// TwinCAT 3 PLC project Tc_Devices
// Title: Tc_Devices
// Company: NewEngineer
// Author: https://github.com/phucpha
// ProjectVersion: 3.2.3.0
// Description: this library use for all Real devices without require special license.
// ProgramVersion: 3.1.4024.0
// libraries:
//   Tc2_Standard, * (Beckhoff Automation GmbH)
//   Tc2_System, * (Beckhoff Automation GmbH)
//   Tc3_Module, * (Beckhoff Automation GmbH)
//   Tc_Utilities, * (NewEngineer)
// project tree:
//   DUTs/ActivePower/ E_ActivePowerType.TcDUT
//   DUTs/Burner/ E_EcoFlamState.TcDUT, E_EcoFlamStateResetV3.TcDUT
//   DUTs/Contactor/ E_ContactorError.TcDUT, E_ContactorState.TcDUT, E_ContactorStateGo.TcDUT
//   DUTs/Cylinder/Universal Cylinder/ E_CylinderError.TcDUT, E_CylinderState.TcDUT, E_CylinderStateGo.TcDUT (not stored)
//   DUTs/Digital Devices/Digital Input/ E_DigitalInputExState.TcDUT (not stored)
//   DUTs/Digital Devices/Lamp Indicator/ E_LampState.TcDUT
//   DUTs/Tank/ E_TankState.TcDUT
//   DUTs/Visu/Burner/ E_VisuCtrlBurnerState.TcDUT, ST_VisuCtrlBurnerFrame.TcDUT
//   DUTs/Visu/Cylinder/ E_VisuCtrlCylinderImgType.TcDUT (not stored), E_VisuCtrlSingleCylinderState.TcDUT (not stored), ST_VisuCtrlCylinderFrame.TcDUT
//   DUTs/Visu/DIDO/ ST_VisuCtrlInputFrame.TcDUT, ST_VisuCtrlOutputFrame.TcDUT
//   / GlobalTextList.TcGTLO, PlcTask.TcTTO
//   POUs/ActivePower/ I_ActivePower.TcIO, I_ActivePowerNoFB.TcIO
//   POUs/AnalogIn/ FB_AnalogInputThermocouple.TcPOU
//   POUs/BurnerEcoflam/ FB_BurnerControlEcoFlam.TcPOU, FB_BurnerControlEcoFlamV2.TcPOU, FB_BurnerControlEcoFlamV3.TcPOU, I_BurnerControlEcoFlam.TcIO, I_BurnerControlEcoFlamV2.TcIO, I_BurnerControlEcoFlamV3.TcIO
//   POUs/ContactorTherRelay/ FB_Contactor1FB_ThermalRelay.TcPOU, FB_ContactorNonFB_Flex_ThermalRelay.TcPOU, FB_ContactorNonFB_ThermalRelay.TcPOU
//   POUs/Contactor/ FB_ContactorFBNO.TcPOU, FB_ContactorNonFB_Flex.TcPOU, FB_ContactorNonFB.TcPOU
//   POUs/Cylinder/Double Coil Cylinder/ FB_DoubleCoilCylinder.TcPOU (not stored)
//   POUs/Cylinder/Single Coil Cylinder/ FB_SingleCoilCylinder.TcPOU (not stored)
//   POUs/Cylinder/Universal Cylinder/ FB_UniversalCylinder.TcPOU, I_UniversalCylinder.TcIO (not stored)
//   POUs/Digital Devices/Digital Device/ FB_DigitalDevice.TcPOU, I_DigitalDevice.TcIO (not stored)
//   POUs/Digital Devices/Digital Input/ FB_DigitalInput.TcPOU, FB_DigitalInputExt.TcPOU, I_DigitalInput.TcIO (not stored)
//   POUs/Digital Devices/Digital Output/ FB_DigitalOutput.TcPOU, I_DigitalOutput.TcIO (not stored)
//   POUs/Digital Devices/Lamp Indicator/ FB_Lamp.TcPOU, I_Lamp.TcIO (not stored)
//   POUs/ POU.TcPOU
//   POUs/Tank0FB/ FB_SingleTankSV1Ext.TcPOU, FB_SingleTankSV1.TcPOU, FB_SingleTankS.TcPOU
//   POUs/TankFB/ FB_SingleTank.TcPOU (not stored), FB_SingleTankV0.TcPOU, FB_SingleTankV1.TcPOU, FB_TankFourCompartments.TcPOU
//   POUs/TankFB/Fill/ FB_TankFill_2Cylinder.TcPOU, I_TankFill.TcIO
//   POUs/TankMix/ FB_Mixer0.TcPOU
//   VISUs/Image Pools/ IPCylinder.TcIPO (not stored)
//   VISUs/Pages/ PageManualCylinders.TcVIS, PageManualInputs.TcVIS, PageManualOutputs.TcVIS, PageManualSafety.TcVIS
//   VISUs/Single/ SingleCylinder.TcVIS, SingleDigitalInput.TcVIS, SingleDigitalOutput.TcVIS, SingleSafeInput.TcVIS, SingleSafeOutput.TcVIS
//   VISUs/Text Lists/ TL_SingleCylinderState.TcTLO
// real-time tasks:
//   TASK PlcTask: cycle T#10ms, priority 20, ADS port 350

CONFIGURATION Tc_Devices
    RESOURCE PLC ON TwinCAT3
        TASK PlcTask(INTERVAL := T#10ms, PRIORITY := 20);
        PROGRAM POU WITH PlcTask : POU;
    END_RESOURCE
END_CONFIGURATION

// ---- DUTs/ActivePower/E_ActivePowerType.TcDUT
{attribute 'strict'}
TYPE E_ActivePowerType :
(
	ACTIVE_POWER_TYPE_NO_FEEDBACK,
	ACTIVE_POWER_TYPE_FEEDBACK
);
END_TYPE

// ---- DUTs/Burner/E_EcoFlamState.TcDUT
{attribute 'strict'}
{attribute 'to_string'}
TYPE E_EcoFlamState :
(
	ECOFLAM_ABORTING := -50,
	ECOFLAM_UNINITIALIZED := 0,
	ECOFLAM_INITIALIZING := 10,
	ECOFLAM_READY_INITIALIZED := 20,
	ECOFLAM_IGNITION := 30,
	ECOFLAM_IGNITION_DONE := 40,
	ECOFLAM_STOP := 50,
	ECOFLAM_STOP_DONE := 60,
	ECOFLAM_RESET := 70,
	ECOFLAM_RESET_DONE := 80
);
END_TYPE

// ---- DUTs/Burner/E_EcoFlamStateResetV3.TcDUT
{attribute 'strict'}
TYPE E_EcoFlamStateResetV3 :
(
	ECOFLAM_V3_RESET_TURN_OFF,
	ECOFLAM_V3_RESET_TURN_ON,
	ECOFLAM_V3_RESET_PORESET_ON
);
END_TYPE

// ---- DUTs/Contactor/E_ContactorError.TcDUT
{attribute 'strict'}
{Attribute 'to_string'}
TYPE E_ContactorError :
(
	CONTACTOR_ERROR_OK := 0,
	CONTACTOR_ERROR_POWER_ON_TIMED_OUT := 20
)UDINT := CONTACTOR_ERROR_OK;
END_TYPE

// ---- DUTs/Contactor/E_ContactorState.TcDUT
{attribute 'strict'}
{Attribute 'to_string'}
TYPE E_ContactorState :
(
	CONTACTOR_ABORTING 			:= -10,
	CONTACTOR_UNINITIALIZED		:= 0,	
	CONTACTOR_INITIALIZING		:= 10,	
	CONTACTOR_READY_INITIALIZED	:= 20,	
	CONTACTOR_IDLE				:= 30,	
	CONTACTOR_POWER_ON			:= 40,
	CONTACTOR_POWER_ON_DONE		:= 50,
	CONTACTOR_POWER_OFF			:= 60,
	CONTACTOR_POWER_OFF_DONE	:= 70,
	CONTACTOR_RESET				:= 100,
	CONTACTOR_RESET_DONE		:= 110

);
END_TYPE

// ---- DUTs/Contactor/E_ContactorStateGo.TcDUT
{Attribute 'to_string'}
{attribute 'strict'}
TYPE E_ContactorStateGo :
(
	CONTACTOR_MOVE_START_TRACKING	:= 0,
	CONTACTOR_MOVE_DELAY			:= 10,
	CONTACTOR_MOVE_DONE				:= 20
);
END_TYPE

// ---- DUTs/Cylinder/Universal Cylinder/E_CylinderError.TcDUT
{attribute 'strict'}
{attribute 'to_string'}
TYPE E_CylinderError :
(
	CYLINDER_ERROR_OK						:= 0,	(*  *)
	CYLINDER_ERROR_MOVE_HOME_TIMED_OUT 		:= 10,	(*  *)
	CYLINDER_ERROR_MOVE_ACTIVE_TIMED_OUT 	:= 20	(*  *)
);
END_TYPE

// ---- DUTs/Cylinder/Universal Cylinder/E_CylinderState.TcDUT
{attribute 'strict'}
{attribute 'to_string'}
TYPE E_CylinderState :
(
	CYLINDER_UNINITIALIZED		:= 0,	(* Cylinder is uninitialized *)
	CYLINDER_INITIALIZING		:= 10,	(* Initialization in progress *)
	CYLINDER_READY_INITIALIZED	:= 20,	(*  *)
	CYLINDER_IDLE				:= 30,	(* Cylinder ready to work *)
	CYLINDER_GO_ACTIVE			:= 40,	(* Cylinder is going to active position *)
	CYLINDER_GO_ACTIVE_DONE		:= 50,	(* Cylinder is in active position *)
	CYLINDER_GO_HOME			:= 60,	(* Cylinder is going to home position *)
	CYLINDER_GO_HOME_DONE		:= 70,	(* Cylinder is in home position *)
	CYLINDER_RELEASE			:= 80,	(* Cylinder is going to release all valves *)
	CYLINDER_RELEASE_DONE		:= 90,	(* Cylinder has been released *)
	CYLINDER_RESET				:= 100,	(* Reseting function block *)
	CYLINDER_RESET_DONE			:= 110,	(* Reset done *)
	CYLINDER_ABORTING 			:= -10	(* Aborting *)
);
END_TYPE

// ---- DUTs/Digital Devices/Lamp Indicator/E_LampState.TcDUT
{attribute 'strict'}
{Attribute 'to_string'}
TYPE E_LampState :
(
	LAMP_OFF 			:= 0,	(* Lamp is off *)
	LAMP_ON				:= 10,	(* Lamp is on *)
	LAMP_BLINKING_OFF	:= 20,	(* Lamp is blinking - current off *)
	LAMP_BLINKING_ON	:= 30	(* Lamp is bliniking - current on *)
);
END_TYPE

// ---- DUTs/Tank/E_TankState.TcDUT
TYPE E_TankState :
(	TANK_IDLE := 0,
	TANK_STOP := 5,
	TANK_WITHDRAWING := 10,
	TANK_WITHDRAWING_DONE := 15,
	TANK_FILLING:= 20
);
END_TYPE

// ---- DUTs/Visu/Burner/E_VisuCtrlBurnerState.TcDUT
{attribute 'strict'}
TYPE E_VisuCtrlBurnerState :
(
	VISU_CTRL_BURNER_WAIT_FOR_CMD 		:= 0,	(* *)
	VISU_CTRL_BURNER_INIT				:= 10,	(*  *)
	VISU_CTRL_BURNER_RESET				:= 20,	(*  *)
	VISU_CTRL_BURNER_IGNITION			:= 30,	(*  *)
	VISU_CTRL_BURNER_STOP				:= 40,	(*  *)
	VISU_CTRL_BURNER_APPEND_POWER_ON	:= 50,	(*  *)	
	VISU_CTRL_BURNER_ABORT				:= -10	(*  *)
);
END_TYPE

// ---- DUTs/Visu/Burner/ST_VisuCtrlBurnerFrame.TcDUT
TYPE ST_VisuCtrlBurnerFrame :
STRUCT
	btnInit				: BOOL;
	btnReset			: BOOL;
	btnAbort			: BOOL;
	btnAppendPowerOn	: BOOL;
	btnIgnition			: BOOL;
	btnStop				: BOOL;
	sName				: STRING;
	bError				: BOOL;
	bFault				: BOOL;
	bIgnitionSuccess	: BOOL;
	
	eState				: E_EcoFlamState;
	sState				: STRING;
END_STRUCT
END_TYPE

// ---- DUTs/Visu/Cylinder/ST_VisuCtrlCylinderFrame.TcDUT
TYPE ST_VisuCtrlCylinderFrame:
STRUCT
	sName			: STRING;
	btnInit				: BOOL;				(*  *)
	btnAbort			: BOOL;				(*  *)
	btnReset			: BOOL;				(*  *)
	btnGoHome 			: BOOL;				(*  *)
	btnGoActive 		: BOOL;				(*  *)
	btnRealase 			: BOOL;				(*  *)
	
	bSensorHome 		: BOOL;				(*  *)
	bSensorActive 		: BOOL;				(*  *)
	bPositionHold		: BOOL;				(*  *)
	bError				: BOOL;				(*  *)
	iErrorID			: UDINT;			(*  *)
	
	tActiveMovement 	: TIME;				(*  *)
	tHomeMovement 		: TIME;				(*  *)
	
	sActiveDescription 	: STRING;			(*  *)
	sHomeDescription 	: STRING;			(*  *)
	sStateDescription	: STRING;			(*  *)
	
	sCylinderImage		: STRING;			(*  *)
	eCylinderState		: E_CylinderState;	(*  *)
	sCylinderState		: STRING;
END_STRUCT
END_TYPE

// ---- DUTs/Visu/DIDO/ST_VisuCtrlInputFrame.TcDUT
TYPE ST_VisuCtrlInputFrame:
STRUCT
	sName			: STRING;
	bIn				: BOOL;								(*  *)
	bForceIn		: BOOL;								(*  *)
	bForceDisabled	: BOOL	:=TRUE ;					(*  *)
	sModuleType		: STRING;							(* Module type e.g. EL1xxx *)
	sPortID			: STRING;							(* Wire id connected to port *)
END_STRUCT
END_TYPE

// ---- DUTs/Visu/DIDO/ST_VisuCtrlOutputFrame.TcDUT
TYPE ST_VisuCtrlOutputFrame:
STRUCT
	sName			: STRING;
	btnOut 			: BOOL; 		(* This button allows to control ouptu manualy if it's set as controlable *)
	bOut 			: BOOL;			(* This bit indicates the status of output in manual mode *)
	bControlable	: BOOL;			(* This bit is used to lock control of output via manual mode - read access only *)
	sModuleType		: STRING;		(* Module type e.g. EL1xxx *)
	sPortID			: STRING;		(* Wire id connected to port *)
END_STRUCT
END_TYPE

// ---- POUs/ActivePower/I_ActivePower.TcIO
INTERFACE I_ActivePower	// don't not EXTENDS I_ActivePowerNoFB, it violates Liskov Substitution Principle (LSP)

PROPERTY Active : reference to bool
GET
END_GET
END_PROPERTY

PROPERTY Busy : REFERENCE TO bool
GET
END_GET
END_PROPERTY

PROPERTY Error : reference to bool
GET
END_GET
END_PROPERTY

METHOD MR_Abort : bool
VAR_INPUT
END_VAR
END_METHOD

METHOD MR_Init : bool
VAR_INPUT
END_VAR
END_METHOD

METHOD MR_PowerOFF : BOOL
VAR_INPUT
END_VAR
END_METHOD

METHOD MR_PowerON : BOOL
VAR_INPUT
END_VAR
END_METHOD

METHOD MR_Reset : bool
VAR_INPUT
END_VAR
END_METHOD

PROPERTY Name : STRING
GET
END_GET
SET
END_SET
END_PROPERTY

(*Powerer on success*)
PROPERTY Powered : REFERENCE TO BOOL
GET
END_GET
END_PROPERTY

PROPERTY PowerOffIsCalled : bool
GET
END_GET
END_PROPERTY

PROPERTY PowerOnIsCalled : bool
GET
END_GET
END_PROPERTY

(*return value depedning on Request*)
PROPERTY ReasonError : string
GET
END_GET
END_PROPERTY

END_INTERFACE

// ---- POUs/ActivePower/I_ActivePowerNoFB.TcIO
INTERFACE I_ActivePowerNoFB

METHOD MR_PowerOFF : BOOL
VAR_INPUT
END_VAR
END_METHOD

METHOD MR_PowerON : BOOL
VAR_INPUT
END_VAR
END_METHOD

PROPERTY Name : STRING
GET
END_GET
SET
END_SET
END_PROPERTY

PROPERTY PowerOffIsCalled : bool
GET
END_GET
END_PROPERTY

PROPERTY PowerOnIsCalled : bool
GET
END_GET
END_PROPERTY

END_INTERFACE

// ---- POUs/BurnerEcoflam/I_BurnerControlEcoFlam.TcIO
INTERFACE I_BurnerControlEcoFlam

PROPERTY Busy : reference to bool
GET
END_GET
END_PROPERTY

PROPERTY Error : REFERENCE to bool
GET
END_GET
END_PROPERTY

PROPERTY IgnitionSucess : bool
GET
END_GET
END_PROPERTY

PROPERTY Inited : bool
GET
END_GET
END_PROPERTY

PROPERTY IsStop : bool
GET
END_GET
END_PROPERTY

METHOD MR_Abort : BOOL
VAR_INPUT
END_VAR
END_METHOD

METHOD MR_AppendPowerOn : BOOL
VAR_INPUT
	iPowerON	: I_ActivePower;
END_VAR
END_METHOD

METHOD MR_Ignition : BOOL
VAR_INPUT
END_VAR
END_METHOD

METHOD  MR_Init : bool // just Acknowledge already append the I_activepower
VAR_INPUT
END_VAR
END_METHOD

METHOD MR_Reset : BOOL
VAR_INPUT
END_VAR
END_METHOD

METHOD MR_Stop : BOOL
VAR_INPUT
END_VAR
END_METHOD

PROPERTY Name : string
GET
END_GET
SET
END_SET
END_PROPERTY

PROPERTY Ref_IfActivePower : REFERENCE TO I_ActivePower
GET
END_GET
END_PROPERTY

PROPERTY Ref_piFault : reference to  FB_DigitalInput
GET
END_GET
END_PROPERTY

PROPERTY Ref_piIgnitionSucess : reference to  FB_DigitalInput
GET
END_GET
END_PROPERTY

PROPERTY State : E_EcoFlamState
GET
END_GET
END_PROPERTY

END_INTERFACE

// ---- POUs/BurnerEcoflam/I_BurnerControlEcoFlamV2.TcIO
INTERFACE I_BurnerControlEcoFlamV2 EXTENDS I_BurnerControlEcoFlam

PROPERTY Ref_poReset : REFERENCE TO fb_digitalOutput
GET
END_GET
END_PROPERTY

END_INTERFACE

// ---- POUs/BurnerEcoflam/I_BurnerControlEcoFlamV3.TcIO
INTERFACE I_BurnerControlEcoFlamV3 EXTENDS I_BurnerControlEcoFlamV2

PROPERTY Ref_poGasLv1 : REFERENCE TO FB_DigitalOutput
GET
END_GET
END_PROPERTY

PROPERTY Ref_poGasLv2 : REFERENCE TO FB_DigitalOutput
GET
END_GET
END_PROPERTY

PROPERTY Ref_poOnOff : REFERENCE TO FB_DigitalOutput
GET
END_GET
END_PROPERTY

END_INTERFACE

// ---- POUs/TankFB/Fill/I_TankFill.TcIO
INTERFACE I_TankFill

METHOD Close : BOOL
VAR_INPUT
END_VAR
END_METHOD

PROPERTY IsClose : bool
GET
END_GET
END_PROPERTY

PROPERTY IsOpen : bool
GET
END_GET
END_PROPERTY

METHOD Open : BOOL
VAR_INPUT
END_VAR
END_METHOD

END_INTERFACE

// ---- POUs/POU.TcPOU
PROGRAM POU
VAR
//	FB_BurnerControlEcoFlam : FB_BurnerControlEcoFlam;
//	FB_BurnerControlEcoFlamV2 : FB_BurnerControlEcoFlamV2;
//	FB_BurnerControlEcoFlamV3 : FB_BurnerControlEcoFlamV3;
//	FB_ContactorFBNO : FB_ContactorFBNO;
//	fb_contactorNonFB : FB_ContactorNonFB;
//	FB_Contactor1FB_ThermalRelay : FB_Contactor1FB_ThermalRelay;
//	FB_ContactorNonFB_ThermalRelay : FB_ContactorNonFB_ThermalRelay;
//	FB_ContactorNonFB_Flex_ThermalRelay : FB_ContactorNonFB_Flex_ThermalRelay;
//	FB_SingleCoilCylinder : FB_SingleCoilCylinder;
//	FB_DoubleCoilCylinder : FB_DoubleCoilCylinder;
//	fbsingletank : FB_SingleTank;
//	fbsingletankV0 : FB_SingleTankV0;
//	fbsingletankV1 : FB_SingleTankV1;
//	fbTankFourCompartments : FB_TankFourCompartments;
//	fbSingleTankV1 : FB_SingleTanksV1;
//	fbFillTank : FB_TankFill_2Cylinder;
//	fbMixer0 : FB_Mixer0;
 	//bIsClose : BOOL;
END_VAR

//fbSingleTankV1.AssignIfill(iFill := fbFillTank);
//bIsClose := fbsingletankV1.Ref_iFill.IsClose;

END_PROGRAM

// ---- POUs/AnalogIn/FB_AnalogInputThermocouple.TcPOU
FUNCTION_BLOCK FB_AnalogInputThermocouple EXTENDS FB_DigitalDevice// use for El 3314
VAR
	iRawValue	AT%I*: INT;
	lrSclale : LREAL := 0.1;
	lrValue	: LREAL;
	bError		AT%I* : BOOL;
	
END_VAR

lrValue := INT_TO_LREAL(iRawValue)*lrSclale;

PROPERTY Error :  bool
GET
Error := bError;
END_GET
END_PROPERTY

PROPERTY Scale : lreal // Value = rawValue form terminal * scale
GET
Scale := lrSclale;
END_GET
SET
lrSclale := Scale;
END_SET
END_PROPERTY

{attribute 'monitoring' := 'variable'}
PROPERTY Value : REFERENCE TO  lreal
GET
Value ref= lrValue;
END_GET
END_PROPERTY

END_FUNCTION_BLOCK

// ---- POUs/Digital Devices/Digital Device/FB_DigitalDevice.TcPOU
(* 
:Description: This function block is base for all other digital devices.
*)
FUNCTION_BLOCK ABSTRACT FB_DigitalDevice IMPLEMENTS I_DigitalDevice
VAR
	sName : STRING; (* Name of digital device instance *)
	sModuleType : STRING;
	sPortID		: STRING;
END_VAR

PROPERTY ModuleType : REFERENCE TO STRING
GET
ModuleType REF= sModuleType;
END_GET
END_PROPERTY

METHOD MR_FirstCycle : BOOL
VAR_INPUT
	sName : STRING;
	sModuleType : STRING;
	sPortID		: STRING;
END_VAR
THIS^.sName := sName;
THIS^.sModuleType := sModuleType;
THIS^.sPortID := sPortID;
END_METHOD

PROPERTY Name : REFERENCE TO STRING
GET
Name REF= sName;
END_GET
END_PROPERTY

PROPERTY PortID : REFERENCE TO STRING
GET
PortID REF= sPortID;
END_GET
END_PROPERTY

END_FUNCTION_BLOCK

// ---- POUs/BurnerEcoflam/FB_BurnerControlEcoFlam.TcPOU
(* This function use for BurnerControlEcoFlam
| this version dont have Reset components like Digital output, user have to reset manual at the BurnerControlEcoFlam device
*)
FUNCTION_BLOCK FB_BurnerControlEcoFlam IMPLEMENTS I_BurnerControlEcoFlam

VAR
	piFault	: FB_DigitalInput;
	piFireSussess : FB_DigitalInputExt;
	ifActivePower : I_ActivePower;					//have FB
	ifActivePowerNoFB : I_ActivePowerNoFB;
	eActivePowerType : E_ActivePowerType;
	eState	: E_EcoFlamState;
	bAbort: BOOL;
	bBusy: BOOL;
	bInit: BOOL;
	bReset: BOOL;
	bStop: BOOL;
	bError : BOOL;
	tMeasurement	: TIME := T#200S;
	bIgnition: BOOL;
	bIgnitioned: BOOL;
	tonMeasurementTimer: Ton;
	tBurnSuccess: TIME;
	sName : STRING;
END_VAR

bError := piFault.In; //OR piFireSussess.ErrorTimedout;
piFireSussess();
StateMachine();
tonMeasurementTimer(PT := tMeasurement);
IF piFireSussess.RisingTrigger AND eState = ECOFLAM_IGNITION THEN
	tBurnSuccess	:= 	tonMeasurementTimer.ET;				
END_IF

PROPERTY ActivePowerType : Reference to E_ActivePowerType
GET
ActivePowerType ref= eActivePowerType;
END_GET
END_PROPERTY

{attribute 'monitoring' := 'variable'}
PROPERTY Busy : reference to bool
GET
Busy ref= bBusy;
END_GET
END_PROPERTY

PROPERTY Error : REFERENCE to bool
GET
error REF= bError;
END_GET
END_PROPERTY

{attribute 'monitoring' := 'variable'}
PROPERTY IgnitionSucess : bool
GET
CASE eActivePowerType OF
	ACTIVE_POWER_TYPE_NO_FEEDBACK:
		IgnitionSucess := piFireSussess.In AND ifActivePowerNoFB.PowerOnIsCalled;
		
	ACTIVE_POWER_TYPE_FEEDBACK:
		IgnitionSucess := piFireSussess.In AND ifActivePower.PowerOnIsCalled;
END_CASE
END_GET
END_PROPERTY

PROPERTY Inited : bool
GET
Inited := eState=ECOFLAM_READY_INITIALIZED;
END_GET
END_PROPERTY

PROPERTY IsRefActivePower : bool
GET
IsRefActivePower := ifActivePower<>0 OR ifActivePowerNoFB<>0;
END_GET
END_PROPERTY

PROPERTY IsStop : bool
GET
CASE eActivePowerType OF
	ACTIVE_POWER_TYPE_NO_FEEDBACK:
		isStop := ifActivePowerNoFB.PowerOffIsCalled;
		
	ACTIVE_POWER_TYPE_FEEDBACK:
		isStop := NOT ifActivePower.Powered;
END_CASE
END_GET
END_PROPERTY

METHOD MR_Abort : BOOL
VAR_INPUT
END_VAR
IF eState >= ECOFLAM_INITIALIZING THEN
	bAbort := TRUE;
	bBusy := TRUE;
	MR_Abort := FALSE;
	eState := ECOFLAM_ABORTING;
ELSIF eState = ECOFLAM_UNINITIALIZED THEN
	bAbort := FALSE;
	bBusy := FALSE;
	MR_Abort := TRUE;
END_IF
END_METHOD

METHOD MR_AppendPowerOn : BOOL
VAR_INPUT
	iPowerON	: I_ActivePower;
END_VAR
IF THIS^.ifActivePower <> iPowerON THEN
	THIS^.ifActivePower := iPowerON;
	MR_AppendPowerOn := true;
END_IF
END_METHOD

METHOD MR_AppendPowerOnNoFB : BOOL
VAR_INPUT
	iPowerOnNoFB	: I_ActivePowerNoFB;
END_VAR
IF THIS^.ifActivePowerNoFB <> iPowerOnNoFB THEN
	THIS^.ifActivePowerNoFB := iPowerOnNoFB;
	MR_AppendPowerOnNoFB := true;
END_IF
END_METHOD

METHOD MR_ChooseIfActivePowerType : BOOL
VAR_INPUT
	eChoseActivePowerType : E_ActivePowerType;
END_VAR
eActivePowerType := eChoseActivePowerType;
END_METHOD

METHOD MR_FirstCycle : BOOL
VAR_INPUT
	sName 							: STRING;
	sPiFireSuccessModuleType		: STRING;
	sPiFirePortID					: STRING;
	sPiFaultModuleType				: STRING;
	sPiFaultPortID					: STRING;
	tONBurnerTimeOut				: TIME;
END_VAR
THIS^.sName := sName;
THIS^.piFireSussess.MR_FirstCycleEx(
 	sName			:= CONCAT(sName,':FireSuccess SS'),
	sModuleType 	:= sPiFireSuccessModuleType,
	sPortID			:= sPiFirePortID,
	bEnableTimeout	:= TRUE,
	tDefaultTimeout	:= tONBurnerTimeOut
);
										
THIS^.piFault.MR_FirstCycle(
	sName := CONCAT(sName,':Fault SS'),
	sModuleType := sPiFaultModuleType,
	sPortID := sPiFaultPortID
);
END_METHOD

METHOD MR_Ignition : BOOL
VAR_INPUT
END_VAR
CASE eActivePowerType OF
	ACTIVE_POWER_TYPE_NO_FEEDBACK:
		IF eState = ECOFLAM_READY_INITIALIZED AND NOT ifActivePowerNoFB.PowerOnIsCalled THEN
			bIgnition	:= TRUE;
			MR_Ignition := FALSE;
			bIgnitioned	:= FALSE;
			eState := ECOFLAM_IGNITION;
			bBusy := TRUE;
		ELSIF eState = ECOFLAM_IGNITION_DONE THEN
			bIgnition := FALSE;
			bIgnitioned	:= TRUE;
			MR_Ignition := TRUE;
			bBusy := false	;
		END_IF
		
	ACTIVE_POWER_TYPE_FEEDBACK:
		IF eState = ECOFLAM_READY_INITIALIZED AND NOT ifActivePower.PowerOnIsCalled THEN
			bIgnition	:= TRUE;
			MR_Ignition := FALSE;
			bIgnitioned	:= FALSE;
			eState := ECOFLAM_IGNITION;
			bBusy := TRUE;
		ELSIF eState = ECOFLAM_IGNITION_DONE THEN
			bIgnition := FALSE;
			bIgnitioned	:= TRUE;
			MR_Ignition := TRUE;
			bBusy := false	;
		END_IF
END_CASE
END_METHOD

METHOD  MR_Init : bool // just Acknowledge already append the I_activepower
VAR_INPUT
END_VAR
IF eState = ECOFLAM_UNINITIALIZED THEN
	bInit := TRUE;
	bBusy := TRUE;
	MR_Init := FALSE;
	eState := ECOFLAM_INITIALIZING;
ELSIF eState = ECOFLAM_READY_INITIALIZED THEN
	bInit := FALSE;
	MR_Init := TRUE;
	bBusy := false;
END_IF
END_METHOD

METHOD MR_Reset : BOOL
VAR_INPUT
END_VAR
IF eState >= ECOFLAM_READY_INITIALIZED AND bError THEN
	bBusy := TRUE;
	bReset := TRUE;
	MR_Reset := FALSE;
	eState := ECOFLAM_RESET;
ELSIF eState = ECOFLAM_RESET_DONE THEN
	bBusy := TRUE;
	bReset := FALSE;
	MR_Reset := TRUE;
END_IF
END_METHOD

METHOD MR_Stop : BOOL
VAR_INPUT
END_VAR
CASE eActivePowerType OF
	ACTIVE_POWER_TYPE_NO_FEEDBACK:
		IF eState >= ECOFLAM_INITIALIZING 
			AND eState < ECOFLAM_STOP_DONE 
			AND ifActivePowerNoFB.PowerOnIsCalled  
		THEN
			bStop := true;
			MR_Stop := FALSE;
			bBusy := TRUE;
			eState := ECOFLAM_STOP;
		ELSIF eState = ECOFLAM_STOP_DONE THEN
			bStop := FALSE;
			MR_Stop := TRUE;
			bBusy := false;
		END_IF 
		
	ACTIVE_POWER_TYPE_FEEDBACK:
		IF eState >= ECOFLAM_INITIALIZING 
			AND eState < ECOFLAM_STOP_DONE 
			AND ifActivePower.Powered  
		THEN
			bStop := true;
			MR_Stop := FALSE;
			bBusy := TRUE;
			eState := ECOFLAM_STOP;
		ELSIF eState = ECOFLAM_STOP_DONE THEN
			bStop := FALSE;
			MR_Stop := TRUE;
			bBusy := false;
		END_IF 
END_CASE
END_METHOD

METHOD PROTECTED  MS_Aborting
CASE eActivePowerType OF
	ACTIVE_POWER_TYPE_NO_FEEDBACK:
		ifActivePowerNoFB.MR_PowerOFF();
		piFireSussess.MR_Abort();
		IF NOT piFireSussess.Active THEN
			eState := ECOFLAM_UNINITIALIZED;
		END_IF
		
	ACTIVE_POWER_TYPE_FEEDBACK:
		ifActivePower.MR_PowerOFF();
		piFireSussess.MR_Abort();
		IF NOT ifActivePower.Powered 
			AND NOT ifActivePower.Busy 
			AND NOT piFireSussess.Active
		THEN
			eState := ECOFLAM_UNINITIALIZED;
		END_IF
END_CASE
END_METHOD

METHOD PROTECTED MS_Ignition
VAR_INPUT
END_VAR
CASE eActivePowerType OF
	ACTIVE_POWER_TYPE_NO_FEEDBACK:
		ifActivePowerNoFB.MR_PowerON();
		piFireSussess.MR_StartTracking();
		tonMeasurementTimer.IN := TRUE;
		IF piFireSussess.In  THEN
			eState := ECOFLAM_IGNITION_DONE;
		END_IF
		
	ACTIVE_POWER_TYPE_FEEDBACK:
		ifActivePower.MR_PowerON();
		piFireSussess.MR_StartTracking();
		tonMeasurementTimer.IN := TRUE;
		IF ifActivePower.Powered AND NOT ifActivePower.Busy 
		AND  piFireSussess.In  THEN
			eState := ECOFLAM_IGNITION_DONE;
		END_IF
END_CASE
END_METHOD

METHOD PROTECTED MS_IgnitionDone : BOOL
VAR_INPUT
END_VAR
tonMeasurementTimer.IN := false;
IF NOT bIgnition THEN
	eState :=  ECOFLAM_READY_INITIALIZED;
END_IF
END_METHOD

METHOD PROTECTED MS_Initializing
piFireSussess.MR_Init();
piFireSussess.EnableTimeout := TRUE;

CASE eActivePowerType OF
	ACTIVE_POWER_TYPE_NO_FEEDBACK:
		IF ifActivePowerNoFB <> 0
			AND piFireSussess.Active
		THEN
			eState := ECOFLAM_READY_INITIALIZED;
		END_IF
		
	ACTIVE_POWER_TYPE_FEEDBACK:
		IF ifActivePower <> 0
			AND piFireSussess.Active
		THEN
			eState := ECOFLAM_READY_INITIALIZED;
		END_IF
END_CASE
END_METHOD

METHOD PROTECTED MS_ReadyInitialized
VAR_INPUT
END_VAR
bBusy := false;
END_METHOD

(*
this version just reset piFireSussess, User have to reset manually at the device
*)
METHOD PROTECTED MS_Reset : BOOL
piFireSussess.MR_Reset();
bInit 		:= FALSE;
bAbort		:= FALSE;
bIgnition 	:= FALSE;
bStop 		:= FALSE;
IF NOT piFireSussess.ErrorTimedout THEN
	eState := ECOFLAM_RESET_DONE;
END_IF
END_METHOD

(* don't not edit*)
METHOD PROTECTED MS_ResetDone
VAR_INPUT
END_VAR
eState := ECOFLAM_READY_INITIALIZED;
END_METHOD

METHOD protected MS_Stop 
VAR_INPUT
END_VAR
CASE eActivePowerType OF
	ACTIVE_POWER_TYPE_NO_FEEDBACK:
		ifActivePowerNoFB.MR_PowerOFF();
		eState := ECOFLAM_STOP_DONE;
		
	ACTIVE_POWER_TYPE_FEEDBACK:
		ifActivePower.MR_PowerOFF();
		IF NOT ifActivePower.Powered AND not ifActivePower.Busy THEN
			eState := ECOFLAM_STOP_DONE;
		END_IF
END_CASE
END_METHOD

METHOD protected Ms_StopDone
VAR_INPUT
END_VAR
IF NOT bStop THEN
	eState := ECOFLAM_READY_INITIALIZED;
END_IF
END_METHOD

METHOD PROTECTED MS_Uninitialized
bBusy := FALSE;

piFireSussess.EnableForce := FALSE;
piFireSussess.EnableTimeout := FALSE;

bInit 		:= FALSE;
bReset		:= FALSE;
bAbort		:= FALSE;
END_METHOD

PROPERTY Name : string
GET
Name := sName;
END_GET
SET
sName := Name;
END_SET
END_PROPERTY

PROPERTY Ref_IfActivePower : REFERENCE TO I_ActivePower
GET
Ref_IfActivePower ref= ifActivePower;
END_GET
END_PROPERTY

PROPERTY Ref_IfActivePowerNoFB : REFERENCE TO I_ActivePowerNoFB
GET
Ref_IfActivePowerNoFB ref= ifActivePowerNoFB;
END_GET
END_PROPERTY

PROPERTY Ref_piFault : reference to  FB_DigitalInput
GET
ref_piFault ref= piFault;
END_GET
END_PROPERTY

PROPERTY Ref_piIgnitionSucess : reference to  FB_DigitalInput
GET
ref_piIgnitionSucess ref= piFireSussess;
END_GET
END_PROPERTY

PROPERTY State : E_EcoFlamState
GET
State := eState;
END_GET
END_PROPERTY

METHOD PROTECTED StateMachine
CASE eState OF
	ECOFLAM_UNINITIALIZED :
		MS_Uninitialized();
		
	ECOFLAM_INITIALIZING	:
		MS_Initializing();
		
	ECOFLAM_READY_INITIALIZED :
		MS_ReadyInitialized();
		
	ECOFLAM_IGNITION	:
		MS_Ignition();
		
	ECOFLAM_IGNITION_DONE	:
		MS_IgnitionDone();
		
	ECOFLAM_STOP		:
		MS_Stop();
		
	ECOFLAM_STOP_DONE	:
		Ms_StopDone();
		
	ECOFLAM_RESET:
		MS_Reset();
		
	ECOFLAM_RESET_DONE:
		MS_ResetDone();
		
	ECOFLAM_ABORTING :
		MS_Aborting();
	
END_CASE
END_METHOD

END_FUNCTION_BLOCK

// ---- POUs/Digital Devices/Digital Input/FB_DigitalInput.TcPOU
(* 
| :Description: This function block represents basic digital input and can be used for creating an instance of signle digital input device like buttons, switches, sensors.
| To get the current status of digital input use "Value" property. To simulate state of the input by software set "Enable Force" parameter and change value via "MR_ResetForceValue" and "MR_SetForceValue" methods.
*)
FUNCTION_BLOCK FB_DigitalInput EXTENDS FB_DigitalDevice IMPLEMENTS I_DigitalInput
VAR
	(* Internal status *)
	bIn				AT %I*	: BOOL;		(* Current value of input *)
	bInForced				: BOOL;		(* Forced value from software *)
	bEnableForce			: BOOL;		(* Enable forcing of the input from software *)
	bRisingTrigger 			: BOOL;		(* Rising trigger of input detected*)
	bFallingTrigger 		: BOOL;		(* Falling trigger of input detected*)
	
	(* Function blocks *)
	rtRisingTrigger 		: R_TRIG;	(* Rising trigger detecting FB*)
	ftFallingTrigger		: F_TRIG;	(* Falling trigger detecting FB*)
END_VAR

PROPERTY EnableForce : BOOL
GET
EnableForce := bEnableForce;
END_GET
SET
bEnableForce := EnableForce;
END_SET
END_PROPERTY

PROPERTY FallingTrigger : BOOL
GET
ftFallingTrigger(CLK := In, Q => bFallingTrigger);
FallingTrigger := bFallingTrigger;
END_GET
END_PROPERTY

PROPERTY In : BOOL
GET
IF NOT bEnableForce THEN
	In := bIn;
ELSE
	In := bInForced;
END_IF
END_GET
END_PROPERTY

METHOD MR_ResetForceValue
IF bEnableForce THEN
	bInForced := FALSE;
	
END_IF
END_METHOD

METHOD MR_SetForceValue
IF bEnableForce THEN
	bInForced := TRUE;
	
END_IF
END_METHOD

PROPERTY RisingTrigger : BOOL
GET
rtRisingTrigger(CLK := In, Q => bRisingTrigger);
RisingTrigger := bRisingTrigger;
END_GET
END_PROPERTY

END_FUNCTION_BLOCK

// ---- POUs/Digital Devices/Digital Input/FB_DigitalInputExt.TcPOU
(* 
| :Description: This function block represents basic digital input and can be used for creating an instance of signle digital input device like buttons, switches, sensors.
| To get the current status of digital input use "Value" property. To simulate state of the input by software set "Enable Force" parameter and change value via "MR_ResetForceValue" and "MR_SetForceValue" methods.
*)
FUNCTION_BLOCK FB_DigitalInputExt EXTENDS FB_DigitalInput
VAR
	(* Internal commands *)
	bInit 				: BOOL;		(*  *)
	bAbort				: BOOL;		(*  *)
	bReset				: BOOL;		(*  *)
	bTimeoutTracking	: BOOL;		(* Watchdog timer control bit *)
	
	(* Internal status *)
	bActive				: BOOL;		(*  *)
	bErrorTimedout		: BOOL;		(* Timeout coccured while waiting for signal *)
	eDigitalInputState	: E_DigitalInputExState;
	
	(*Internal parameters*)
	tTimeout			: TIME;		(* Input timeout *)
	bEnableTimeout		: BOOL;		(* Enable using timeout *)
	
	(* Function blocks *)
	bStartWatchdog		: BOOL;
	tonWatchdog			: TON;		(* Input timeout watchdog *)
	
END_VAR

bActive := eDigitalInputState >= DIGITAL_INPUT_EX_IDLE; //OR eDigitalInputState = DIGITAL_INPUT_EX_ABORTING;

StateMachine();

tonWatchdog( IN := bStartWatchdog, PT := tTimeout);

PROPERTY Active : REFERENCE TO BOOL
GET
Active REF= bActive;
END_GET
END_PROPERTY

PROPERTY CurrentTimeout : REFERENCE TO TIME
GET
CurrentTimeout REF= tonWatchdog.ET;
END_GET
END_PROPERTY

PROPERTY EnableTimeout : BOOL
GET
EnableTimeout := bEnableTimeout;
END_GET
SET
bEnableTimeout := EnableTimeout;
END_SET
END_PROPERTY

PROPERTY ErrorTimedout : REFERENCE TO BOOL
GET
ErrorTimedout REF= bErrorTimedout;
END_GET
END_PROPERTY

METHOD MR_Abort : BOOL
VAR_INPUT
END_VAR
IF eDigitalInputState > DIGITAL_INPUT_EX_UNINITIALIZED THEN
	bAbort := TRUE;
	MR_Abort := FALSE;
	eDigitalInputState := DIGITAL_INPUT_EX_ABORTING;
	fbMachineLogger.MR_AddLogs(CONCAT(sName,' : abort requested'));	
	
ELSIF eDigitalInputState = DIGITAL_INPUT_EX_UNINITIALIZED THEN
	bAbort := FALSE;
	MR_Abort := TRUE;
	fbMachineLogger.MR_AddLogs(CONCAT(sName,' : abort done'));	
	
END_IF
END_METHOD

METHOD MR_FirstCycleEx : BOOL
VAR_INPUT
	sName			: STRING;
	sModuleType		: STRING;
	sPortID			: STRING;
	bEnableTimeout	: BOOL;
	tDefaultTimeout : TIME;
END_VAR
THIS^.sName := sName;
THIS^.ModuleType := sModuleType;
THIS^.PortID := sPortID;
THIS^.bEnableTimeout := bEnableTimeout;
THIS^.tTimeout := tDefaultTimeout;
END_METHOD

METHOD MR_Init : BOOL
VAR_INPUT
END_VAR
IF eDigitalInputState = DIGITAL_INPUT_EX_UNINITIALIZED THEN
	bInit := TRUE;
	MR_Init := FALSE;
	eDigitalInputState := DIGITAL_INPUT_EX_INITIALIZING;
	fbMachineLogger.MR_AddLogs(CONCAT(sName,' : initialization requested'));		
	
ELSIF eDigitalInputState = DIGITAL_INPUT_EX_IDLE AND bInit THEN
	bInit := FALSE;
	MR_Init := TRUE;
	fbMachineLogger.MR_AddLogs(CONCAT(sName,' : initialization done'));	

END_IF
END_METHOD

METHOD MR_Reset : BOOL
VAR_INPUT
END_VAR
IF eDigitalInputState = DIGITAL_INPUT_EX_IDLE THEN
	bReset := TRUE;
	MR_Reset := FALSE;
	eDigitalInputState := DIGITAL_INPUT_EX_RESET;
	fbMachineLogger.MR_AddLogs(CONCAT(sName,' : reset requested'));	
	
ELSIF eDigitalInputState = DIGITAL_INPUT_EX_RESET_DONE THEN
	bReset := FALSE;
	MR_Reset := TRUE;
	fbMachineLogger.MR_AddLogs(CONCAT(sName,' : reset done'));	
	
END_IF
END_METHOD

METHOD MR_StartTracking
VAR_INPUT
END_VAR
IF eDigitalInputState = DIGITAL_INPUT_EX_IDLE AND bEnableTimeout AND NOT bErrorTimedout THEN
	bTimeoutTracking := TRUE;
	eDigitalInputState := DIGITAL_INPUT_EX_TIMEOUT_TRACKING;
	fbMachineLogger.MR_AddLogs(CONCAT(sName,' : start tracking requested'));	
	
END_IF
END_METHOD

METHOD PROTECTED MS_Abort
VAR_INPUT
END_VAR
eDigitalInputState := DIGITAL_INPUT_EX_UNINITIALIZED;
END_METHOD

METHOD PROTECTED MS_Idle
VAR_INPUT
END_VAR
;
END_METHOD

METHOD PROTECTED MS_Initializing
VAR_INPUT
END_VAR
(* To-Do add alarm declaration *)

eDigitalInputState := DIGITAL_INPUT_EX_READY_INITIALIZED;
END_METHOD

METHOD PROTECTED MS_ReadyInitialized
VAR_INPUT
END_VAR
eDigitalInputState := DIGITAL_INPUT_EX_IDLE;
END_METHOD

METHOD PROTECTED MS_Reset
VAR_INPUT
END_VAR
bErrorTimedout := FALSE;
eDigitalInputState := DIGITAL_INPUT_EX_RESET_DONE;
END_METHOD

METHOD PROTECTED MS_ResetDone
VAR_INPUT
END_VAR
IF NOT bReset THEN
	eDigitalInputState := DIGITAL_INPUT_EX_IDLE;
END_IF
END_METHOD

METHOD PROTECTED MS_TimeoutTracking
VAR_INPUT
END_VAR
IF tonWatchdog.Q THEN
	(* To-Do raise alarm *)
	bErrorTimedout := TRUE;
	bStartWatchdog := FALSE;
	eDigitalInputState := DIGITAL_INPUT_EX_TIMEOUT_TRACKING_DONE;
	
ELSE
	bStartWatchdog := TRUE;
	
	IF bRisingTrigger OR bFallingTrigger THEN
		bStartWatchdog := FALSE;
		eDigitalInputState := DIGITAL_INPUT_EX_TIMEOUT_TRACKING_DONE;
	
	END_IF
END_IF
END_METHOD

METHOD PROTECTED MS_TimeoutTrackingDone
VAR_INPUT
END_VAR
bTimeoutTracking := FALSE;
eDigitalInputState := DIGITAL_INPUT_EX_IDLE;
END_METHOD

METHOD PROTECTED MS_Uninitialized
VAR_INPUT
END_VAR
bInit := FALSE;
bAbort := FALSE;
bReset := FALSE;
bTimeoutTracking := FALSE;

bRisingTrigger := FALSE;
bFallingTrigger := FALSE;
bErrorTimedout := FALSE;

tonWatchdog( IN := FALSE, PT := tTimeout);
END_METHOD

PROPERTY State : REFERENCE TO E_DigitalInputExState
GET
State REF= eDigitalInputState;
END_GET
END_PROPERTY

METHOD PROTECTED StateMachine
VAR_INPUT
END_VAR
CASE eDigitalInputState OF
	DIGITAL_INPUT_EX_UNINITIALIZED:
		MS_Uninitialized();
		
	DIGITAL_INPUT_EX_INITIALIZING:
		MS_Initializing();
		
	DIGITAL_INPUT_EX_READY_INITIALIZED:
		MS_ReadyInitialized();
		
	DIGITAL_INPUT_EX_IDLE:
		MS_Idle();
		
	DIGITAL_INPUT_EX_TIMEOUT_TRACKING:
		MS_TimeoutTracking();	
	
	DIGITAL_INPUT_EX_TIMEOUT_TRACKING_DONE:
		MS_TimeoutTrackingDone();	
	
	DIGITAL_INPUT_EX_RESET:
		MS_Reset();

	DIGITAL_INPUT_EX_RESET_DONE:
		MS_ResetDone();
	
	DIGITAL_INPUT_EX_ABORTING:
		MS_Abort();
	
END_CASE
END_METHOD

PROPERTY Timeout : TIME
GET
Timeout := tTimeout;
END_GET
SET
tTimeout := Timeout;
END_SET
END_PROPERTY

END_FUNCTION_BLOCK

// ---- POUs/BurnerEcoflam/FB_BurnerControlEcoFlamV2.TcPOU
(* This function use for BurnerControlEcoFlam have Reset by Digital output.
*)
FUNCTION_BLOCK FB_BurnerControlEcoFlamV2 EXTENDS FB_BurnerControlEcoFlam IMPLEMENTS I_BurnerControlEcoFlamV2
VAR
	poReset : FB_DigitalOutput;
	tonReset : TON;
	timeReset : TIME := T#1.5s;
END_VAR

tonReset(
	in := eState=ECOFLAM_RESET,
	PT := timeReset
);
poReset();
poReset.Out := tonReset.IN;
SUPER^();

METHOD PROTECTED MS_Reset : BOOL
piFireSussess.MR_Reset();
bInit 		:= FALSE;
bAbort		:= FALSE;
bIgnition 	:= FALSE;
bStop 		:= FALSE;
IF NOT piFireSussess.ErrorTimedout// for sure least than TimeReset.
	AND tonReset.Q
THEN
	eState := ECOFLAM_RESET_DONE;
END_IF
END_METHOD

PROPERTY Ref_poReset : Reference to FB_DigitalOutput
GET
Ref_poReset ref= poReset;
END_GET
END_PROPERTY

END_FUNCTION_BLOCK

// ---- POUs/Digital Devices/Digital Output/FB_DigitalOutput.TcPOU
(* 
| :Description: This function block represents basic digital output and can be used for creating an instance of signle digital output device. 
| To control the output state use property "Out" 
*)
FUNCTION_BLOCK FB_DigitalOutput EXTENDS FB_DigitalDevice IMPLEMENTS  I_DigitalOutput
VAR
	bOut AT %Q*: BOOL; (* Current value of output*)
END_VAR

PROPERTY Out : BOOL
GET
Out := bOut;
END_GET
SET
bOut := Out;
END_SET
END_PROPERTY

END_FUNCTION_BLOCK

// ---- POUs/BurnerEcoflam/FB_BurnerControlEcoFlamV3.TcPOU
(* this fb for burner type that request off power and turn on again to reset it*)
FUNCTION_BLOCK FB_BurnerControlEcoFlamV3 EXTENDS FB_BurnerControlEcoFlamV2 IMPLEMENTS I_BurnerControlEcoFlamV3
VAR
	poOnOff : FB_DigitalOutput;
	poGasLv1 : FB_DigitalOutput;
	poGasLv2 : FB_DigitalOutput;
	eResetState : E_EcoFlamStateResetV3;
	tonDelayOffPower : TON;
	tonDelayOnPower : TON;
	timeDelayOnOffPower : TIME := T#2S;
END_VAR

IF IsRefActivePower THEN
	CASE ActivePowerType OF
		ACTIVE_POWER_TYPE_FEEDBACK:
			poOnOff.Out := ifActivePower.PowerOnIsCalled;
			poGasLv1.Out := ifActivePower.PowerOnIsCalled;
		ACTIVE_POWER_TYPE_NO_FEEDBACK:
			poOnOff.Out := ifActivePowerNoFB.PowerOnIsCalled;
			poGasLv1.Out := ifActivePowerNoFB.PowerOnIsCalled;
	END_CASE
END_IF
bError := piFault.In;
piFireSussess();
StateMachine();
tonMeasurementTimer(PT := tMeasurement);
IF piFireSussess.RisingTrigger AND eState=ECOFLAM_IGNITION THEN
	tBurnSuccess	:= 	tonMeasurementTimer.ET;				
END_IF

tonReset(
	in := (eState=ECOFLAM_RESET AND eResetState=ECOFLAM_V3_RESET_PORESET_ON),
	PT := timeReset
);
poReset();
poReset.Out := tonReset.IN;
tonDelayOffPower(
	IN := eState=ECOFLAM_RESET AND eresetstate=ECOFLAM_V3_RESET_TURN_OFF,
	PT := timeDelayOnOffPower
);
tonDelayOnPower(
	IN := eState=ECOFLAM_RESET AND eresetstate=ECOFLAM_V3_RESET_TURN_ON,
	PT := timeDelayOnOffPower
);

METHOD PROTECTED MS_Aborting
VAR_INPUT
END_VAR
SUPER^.MS_Aborting();
eResetState := ECOFLAM_V3_RESET_TURN_OFF;
END_METHOD

METHOD PROTECTED MS_Reset : BOOL
piFireSussess.MR_Reset();
bInit 		:= FALSE;
bAbort		:= FALSE;
bIgnition 	:= FALSE;
bStop 		:= FALSE;

CASE eResetState OF
	ECOFLAM_V3_RESET_TURN_OFF:
		CASE THIS^.eActivePowerType OF
			ACTIVE_POWER_TYPE_NO_FEEDBACK:
				ifActivePowerNoFB.MR_PowerOFF();
				IF tonDelayOffPower.Q THEN
					eResetState := ECOFLAM_V3_RESET_TURN_ON;
				END_IF
			ACTIVE_POWER_TYPE_FEEDBACK:
				ifActivePower.MR_PowerOFF();
				IF tonDelayOffPower.Q
					AND NOT ifActivePower.Powered AND NOT ifActivePower.Busy
				THEN
					eResetState := ECOFLAM_V3_RESET_TURN_ON;
				END_IF
		END_CASE
		
	ECOFLAM_V3_RESET_TURN_ON:
		CASE THIS^.eActivePowerType OF
			ACTIVE_POWER_TYPE_NO_FEEDBACK:
				ifActivePowerNoFB.MR_PowerON();
				IF tonDelayOnPower.Q THEN
					eResetState := ECOFLAM_V3_RESET_PORESET_ON;
				END_IF
			ACTIVE_POWER_TYPE_FEEDBACK:
				ifActivePower.MR_PowerON();
				IF (ifActivePower.Powered AND NOT ifActivePower.Busy)
					AND tonDelayOnPower.Q
				THEN
					eResetState := ECOFLAM_V3_RESET_PORESET_ON;
				END_IF
		END_CASE
		
	ECOFLAM_V3_RESET_PORESET_ON:
		IF tonReset.Q THEN
			eState := ECOFLAM_RESET_DONE;
		END_IF
END_CASE
END_METHOD

METHOD PROTECTED MS_ResetDone
VAR_INPUT
END_VAR
SUPER^.MS_ResetDone();
eResetState := ECOFLAM_V3_RESET_TURN_OFF;
END_METHOD

PROPERTY Ref_poGasLv1 : REFERENCE TO FB_DigitalOutput
GET
Ref_poGasLv1 ref= poGasLv1;
END_GET
END_PROPERTY

PROPERTY Ref_poGasLv2 : REFERENCE TO FB_DigitalOutput
GET
Ref_poGasLv2 ref= poGasLv2;
END_GET
END_PROPERTY

PROPERTY Ref_poOnOff : REFERENCE TO FB_DigitalOutput
GET
Ref_poOnOff ref= poOnOff;
END_GET
END_PROPERTY

END_FUNCTION_BLOCK

// ---- POUs/ContactorTherRelay/FB_Contactor1FB_ThermalRelay.TcPOU
(* 
| :Description: this function block is the Contactor FeedbackNO + thermal relay connect toghther.
| Then wiring have to series by Digital output to NC thermal relay to Coil
*)
FUNCTION_BLOCK FB_Contactor1FB_ThermalRelay EXTENDS FB_ContactorFBNO IMPLEMENTS I_ActivePower

VAR
	piFR		: FB_DigitalInput;// thermal relay NO
	bOverload	: BOOL;
END_VAR

bOverload :=  piFR.In;
SUPER^();

PROPERTY IsOverload : REFERENCE to bool
GET
isOverload ref= bOverload;
END_GET
END_PROPERTY

PROPERTY ReasonError : string
GET
IF isOverload THEN 
	ReasonError := 'ThermalRelay OverLoad';
ELSE
	ReasonError := 'Coil of Contactor or NO contact work incorrectly';
END_IF
END_GET
END_PROPERTY

PROPERTY Ref_piFR : reference to FB_DigitalInput
GET
Ref_piFR ref= piFR;
END_GET
END_PROPERTY

END_FUNCTION_BLOCK

// ---- POUs/Contactor/FB_ContactorFBNO.TcPOU
(* 
| :Description: This function block use for Contactor active by digital output, Use NO contact feedback(Digital Input) to Check Error
| Don't not extend the FB_ContactorNonFB because it violate Liskov Substitution Principle (LSP)
*)
FUNCTION_BLOCK FB_ContactorFBNO IMPLEMENTS I_ActivePower
VAR
	piNO 		: FB_DigitalInputExt;
	poCoil		: FB_DigitalOutput;
	sName		: STRING;
	(* Internal commands *)
	bInit 				: BOOL;					(* Prepare contactor to work *)
	bReset				: BOOL;					(* Reset function block *)
	bAbort				: BOOL;					(* Deinitialize function block *)
	bPowerOn			: BOOL;					(* Power On Request *)
	bPowerOff			: BOOL;					(* Power Off Request *)
	bSimulation			: BOOL;					(* Simulation on/off bit *)
	(* Cylinder state *)
	bActive				: BOOL;					(*  *)
	bBusy				: BOOL;					(*  *)	
	bError 				: BOOL;					(*  *)
	bPowered			: BOOL;					(*  *)
	eErrorID 			: E_ContactorError;		(*  *)
	eContactorState		: E_ContactorState;		(* State machine of function block *)
	eContactorGoHomeState : E_ContactorStateGo;
	eContactorGoActiveState : E_ContactorStateGo;
	sReasonError		: STRING;
	(* Timers *)
	tonPowerOnDelay		: TON;					(* Timer ON delay when Power ON Request *)
	tonPowerOffDelay	: TON;					(* Timer OFF delay when Power ON Request *)
	tonMeasurementTimer	: TON;					(* Measurement of movement time *)
	tonContactorWatchdog: TON;					(* Movement watchdog *)
	tonGeneral 			: TON;
	
	(* Time parameters *)
	tDelay				: TIME := T#100MS;		(* Delay time when moving to any position *)
	tMeasurement		: TIME := T#60S;		(* Time of movement measurement *)
	tPowerOn			: TIME;					(* Time of last movement to active postion *)

	
END_VAR
(*
Version history:

+-------------+------------+----------------+-------------------------------+------------------------------------------+
|Date         | Version    | created under  | Author   						| Remark                                   |
+=============+============+================+===============================+==========================================+
|2025-06      | 0.1.1.1   | V3.1.4024.56   | https://github.com/phucpha    | Function block created                   |
+-------------+------------+----------------+-------------------------------+------------------------------------------+

*)

(* Simulation enabled*)
IF bSimulation THEN
	piNO.EnableForce := TRUE;
	M_SimulationLogic();
ELSE
	piNO.MR_ResetForceValue();
	piNO.EnableForce := FALSE;
END_IF

(* Time  measurement - to active position *)
IF piNO.RisingTrigger 
	AND eContactorState = CONTACTOR_POWER_ON
THEN
	tPowerOn := tonMeasurementTimer.ET;
END_IF

(*  *)
tonMeasurementTimer(
	IN := tonContactorWatchdog.IN,
	PT := tMeasurement
);
						
StateMachine();

(* Update status flags *)
bActive := eContactorState >= CONTACTOR_IDLE 
			OR econtactorState = CONTACTOR_ABORTING ;

bError := piNO.ErrorTimedout;

(* Error handling *)
IF piNO.ErrorTimedout THEN
	eErrorID := CONTACTOR_ERROR_POWER_ON_TIMED_OUT;
	fbMachineLogger.MR_AddLogs(
		FUN_MergeStrings5(
			sName,
			' : Error occured (error ID: ',
			'Power On timed out', ')',
			''
		)
	);
ELSE
	eErrorID := CONTACTOR_ERROR_OK;
END_IF

(* Position flag update *)
bPowered := piNO.In;

(* Run sensors instances *)
piNO();
poCoil();

PROPERTY Active : REFERENCE to bool
GET
Active ref= bActive;
END_GET
END_PROPERTY

PROPERTY Busy : REFERENCE TO BOOL
GET
Busy ref= bBusy;
END_GET
END_PROPERTY

PROPERTY Delay : TIME
GET
delay := tDelay;
END_GET
SET
tDelay := Delay;
END_SET
END_PROPERTY

PROPERTY Error : REFERENCE TO BOOL
GET
Error ref= bError;
END_GET
END_PROPERTY

PROPERTY ErrorID : REFERENCE TO UDINT
GET
ErrorID ref= eErrorID;
END_GET
END_PROPERTY

METHOD PROTECTED M_SimulationLogic 
VAR_INPUT
END_VAR
IF poCoil.Out THEN
	piNO.MR_SetForceValue();
	
ELSIF NOT poCoil.Out THEN
	piNO.MR_ResetForceValue();
	
END_IF
END_METHOD

METHOD MR_Abort : BOOL
VAR_INPUT
END_VAR
IF eContactorState >= CONTACTOR_IDLE THEN
	bBusy := TRUE;
	bAbort := TRUE;
	MR_Abort := FALSE;
	eContactorState := CONTACTOR_ABORTING;
	fbMachineLogger.MR_AddLogs(CONCAT(sName,' : abort requested'));	
	
ELSIF eContactorState = CONTACTOR_UNINITIALIZED THEN
	bAbort := FALSE;
	MR_Abort := TRUE;
	fbMachineLogger.MR_AddLogs(CONCAT(sName,' : abort done'));	
	
END_IF
END_METHOD

METHOD MR_FirstCycle : BOOL
VAR_INPUT
	sName 							: STRING;
	sCoilModuleType					: STRING;
	sCoilPortID						: STRING;
	sNOModuleType					: STRING;
	sNOPortID						: STRING;
	tGoActiveTimeout				: TIME;
	tDelay							: TIME;
END_VAR
piNO.EnableTimeout := TRUE;
THIS^.sName := sName;								
THIS^.tDelay := tDelay;	
THIS^.PowerOnTimeout := tGoActiveTimeout;	
THIS^.piNO.MR_FirstCycleEx(
	sName := CONCAT(sName,':NO'),
	sModuleType := sNOModuleType,
	sPortID	:= sNOPortID,
	bEnableTimeout := TRUE,
	tDefaultTimeout	:= tGoActiveTimeout
);
THIS^.poCoil.MR_FirstCycle(
	sName := CONCAT(sName,':Coil'),
	sModuleType := sCoilModuleType,
	sPortID := sCoilPortID
);
END_METHOD

METHOD MR_Init : BOOL
IF eContactorState = CONTACTOR_UNINITIALIZED THEN
	bBusy := TRUE;
	bInit := TRUE;
	MR_Init := FALSE;
	eContactorState := CONTACTOR_INITIALIZING;
	fbMachineLogger.MR_AddLogs(CONCAT(sName,' : initialization requested'));	
	
ELSIF eContactorState = CONTACTOR_IDLE THEN
	bInit := FALSE;
	MR_Init := TRUE;
	fbMachineLogger.MR_AddLogs(CONCAT(sName,' : initialization done'));	
	
END_IF
END_METHOD

METHOD MR_PowerOFF : BOOL
IF eContactorState >= CONTACTOR_IDLE 
	AND eContactorState <= CONTACTOR_POWER_ON_DONE
	AND (piNO.In OR poCoil.Out)
THEN
	bBusy := TRUE;
	bPowerOff := TRUE;
	MR_PowerOFF := FALSE;
	eContactorState := CONTACTOR_POWER_OFF;
	eContactorGoHomeState := CONTACTOR_MOVE_START_TRACKING;
	fbMachineLogger.MR_AddLogs(CONCAT(sName,' :Power Off requested'));	
	
ELSIF eContactorState = CONTACTOR_POWER_OFF_DONE THEN
	bPowerOff := FALSE;
	MR_PowerOFF := TRUE;
	fbMachineLogger.MR_AddLogs(CONCAT(sName,' :Power Off done'));	
END_IF
END_METHOD

METHOD MR_PowerON : BOOL
IF eContactorState = CONTACTOR_IDLE
	AND NOT piNO.In 
THEN
	bBusy := TRUE;
	bPowerOn := TRUE;
	MR_PowerON := FALSE;
	eContactorState := CONTACTOR_POWER_ON;
	eContactorGoActiveState := CONTACTOR_MOVE_START_TRACKING;
	fbMachineLogger.MR_AddLogs(CONCAT(sName,' : Power On requested'));	
	
ELSIF eContactorState = CONTACTOR_POWER_ON_DONE THEN
	bPowerOn := FALSE;
	MR_PowerON := TRUE;
	fbMachineLogger.MR_AddLogs(CONCAT(sName,' : Power On  done'));		
	
END_IF
END_METHOD

METHOD MR_Reset : BOOL
IF eContactorState >= CONTACTOR_IDLE
	AND bError 
THEN
	bBusy := TRUE;
	bReset := TRUE;
	MR_Reset := FALSE;
	eContactorState := CONTACTOR_RESET;
	fbMachineLogger.MR_AddLogs(CONCAT(sName,' : reset requested'));	
	
ELSIF eContactorState = CONTACTOR_RESET_DONE THEN
	bReset := FALSE;
	MR_Reset := TRUE;
	fbMachineLogger.MR_AddLogs(CONCAT(sName,' : reset done'));		
	
END_IF
END_METHOD

METHOD PROTECTED  MS_Aborting
piNO.MR_Abort();

IF  NOT piNO.Active THEN
	//bBusy := FALSE;
	eContactorState := CONTACTOR_UNINITIALIZED;	
END_IF
END_METHOD

METHOD PROTECTED MS_Idle
;
END_METHOD

METHOD PROTECTED MS_Initializing
piNO.MR_Init();
piNO.EnableTimeout := TRUE;

IF piNO.Active 
	AND NOT piNO.In 
THEN
	eCONTACTORState := CONTACTOR_READY_INITIALIZED;
END_IF
tonGeneral(
	in := TRUE,
	pt := T#0.1S
);
IF tonGeneral.Q
	AND piNO.In
THEN
	bError := TRUE;
	sReasonError := 'Coil not active Or NO incorrect';
	tonGeneral(IN := FALSE);
END_IF
END_METHOD

METHOD PROTECTED  MS_PowerOff
bPowerOn := FALSE;
poCoil.Out := FALSE;
CASE eContactorGoHomeState OF
	CONTACTOR_MOVE_START_TRACKING:
		
		IF NOT piNO.In THEN
			IF TIME_TO_INT(tDelay) = 0 THEN
				eContactorGoHomeState := CONTACTOR_MOVE_DONE;
			ELSE
				eContactorGoHomeState := CONTACTOR_MOVE_DELAY;
			END_IF
		END_IF
		
	CONTACTOR_MOVE_DELAY:
		tonPowerOffDelay(IN := TRUE, PT := tDelay);
		
		IF tonPowerOffDelay.Q THEN
			tonPowerOffDelay(IN := FALSE);
			eContactorGoHomeState := CONTACTOR_MOVE_DONE;
		END_IF
		
	CONTACTOR_MOVE_DONE:
		eContactorState := CONTACTOR_POWER_OFF_DONE;
	
END_CASE
END_METHOD

METHOD PROTECTED MS_PowerOffDone
IF NOT bPowerOff THEN
	bBusy := FALSE;
	eContactorState := CONTACTOR_IDLE;
END_IF
END_METHOD

METHOD PROTECTED  MS_PowerOn
poCoil.Out := TRUE;

CASE eContactorGoActiveState OF
	CONTACTOR_MOVE_START_TRACKING:
		piNO.MR_StartTracking();
		
		IF piNO.In THEN
			IF TIME_TO_INT(tDelay) = 0 THEN
				eContactorGoActiveState := CONTACTOR_MOVE_DONE;
			ELSE
				eContactorGoActiveState := CONTACTOR_MOVE_DELAY;
			END_IF
		END_IF
		
	CONTACTOR_MOVE_DELAY:
		tonPowerOnDelay(IN := TRUE, PT := tDelay);
		
		IF tonPowerOnDelay.Q THEN
			tonPowerOnDelay(IN := FALSE);
			eContactorGoActiveState := CONTACTOR_MOVE_DONE;
		END_IF
		
	CONTACTOR_MOVE_DONE:
		eContactorState := CONTACTOR_POWER_ON_DONE;
		
END_CASE
END_METHOD

METHOD PROTECTED MS_PowerOnDone
IF NOT bPowerOn THEN
	bBusy := FALSE;
	eCONTACTORState := CONTACTOR_IDLE;
END_IF
END_METHOD

METHOD PROTECTED MS_ReadyInitialized
VAR_INPUT
END_VAR
bBusy := FALSE;
eContactorState := CONTACTOR_IDLE;
END_METHOD

METHOD PROTECTED MS_Reset
VAR_INPUT
END_VAR
poCoil.Out := FALSE;
bInit 		:= FALSE;
bPowerOn 	:= FALSE;
bPowerOff 	:= FALSE;
bAbort		:= FALSE;
tonPowerOffDelay(IN := FALSE);
tonPowerOnDelay(IN := FALSE);
tonMeasurementTimer(IN:= FALSE);

piNO.MR_Reset();

IF NOT piNO.ErrorTimedout THEN
	eContactorState := CONTACTOR_RESET_DONE;
END_IF
END_METHOD

METHOD PROTECTED MS_ResetDone
VAR_INPUT
END_VAR
IF NOT bReset THEN
	bBusy := FALSE;
	eContactorState := CONTACTOR_IDLE;
END_IF
END_METHOD

METHOD PROTECTED MS_Uninitialized
poCoil.Out := FALSE;

bError := FALSE;
bBusy := FALSE;
bPowered := FALSE;
piNO.EnableForce := FALSE;
piNO.EnableTimeout := FALSE;

bInit 		:= FALSE;
bPowerOn 	:= FALSE;
bPowerOff	:= FALSE;
bReset		:= FALSE;
bAbort		:= FALSE;
sReasonError := '';
tonPowerOnDelay(IN := FALSE);
tonPowerOffDelay(IN := FALSE);
tonMeasurementTimer(IN:= FALSE);
END_METHOD

PROPERTY Name : STRING
GET
name := sName;
END_GET
SET
sName := Name;
END_SET
END_PROPERTY

PROPERTY Powered : REFERENCE TO BOOL
GET
Powered ref= bPowered;
END_GET
END_PROPERTY

PROPERTY PowerOffIsCalled : bool
GET
PowerOffIsCalled := poCoil.Out=FALSE;
END_GET
END_PROPERTY

PROPERTY PowerOnIsCalled : bool
GET
PowerOnIsCalled := poCoil.Out=TRUE;
END_GET
END_PROPERTY

PROPERTY PowerOnTime : REFERENCE TO TIME
GET
PowerOnTime REF= tPowerOn;
END_GET
END_PROPERTY

PROPERTY PowerOnTimeout : TIME
GET
PowerOnTimeout := piNO.Timeout;
END_GET
SET
piNO.Timeout := PowerOnTimeout;
END_SET
END_PROPERTY

(*if Fail*)
PROPERTY ReasonError : string
GET
ReasonError := 'Dont have NO signal when PowerOn';
END_GET
END_PROPERTY

PROPERTY Ref_piNO : reference to  FB_DigitalInput
GET
ref_piNO ref= THIS^.piNO;
END_GET
END_PROPERTY

PROPERTY Ref_poCoil : reference to fb_digitalOutput
GET
ref_poCoil ref= poCoil;
END_GET
END_PROPERTY

PROPERTY Simulation : BOOL
GET
Simulation := bSimulation;
END_GET
SET
bSimulation := Simulation;
END_SET
END_PROPERTY

PROPERTY State : REFERENCE TO E_ContactorState
GET
State ref= THIS^.eContactorState;
END_GET
END_PROPERTY

METHOD PROTECTED StateMachine : BOOL
VAR_INPUT
END_VAR
CASE eContactorState OF
	CONTACTOR_UNINITIALIZED:
		MS_Uninitialized();
		
    CONTACTOR_INITIALIZING:
		MS_Initializing();
		
    CONTACTOR_READY_INITIALIZED:
		MS_ReadyInitialized();
		
    CONTACTOR_IDLE:
		MS_Idle();
				
    CONTACTOR_POWER_ON:
		MS_PowerOn();
			
    CONTACTOR_POWER_ON_DONE:
		MS_PowerOnDone();
	
    CONTACTOR_POWER_OFF:
		MS_PowerOff();
			
    CONTACTOR_POWER_OFF_DONE:
		MS_PowerOffDone();
		
    CONTACTOR_RESET:
		MS_Reset();
				
    CONTACTOR_RESET_DONE:
		MS_ResetDone();
				
    CONTACTOR_ABORTING:			
    	MS_Aborting();

END_CASE
END_METHOD

END_FUNCTION_BLOCK

// ---- POUs/ContactorTherRelay/FB_ContactorNonFB_Flex_ThermalRelay.TcPOU
FUNCTION_BLOCK FB_ContactorNonFB_Flex_ThermalRelay EXTENDS FB_ContactorNonFB_Flex
VAR
	piFR		: FB_DigitalInput;// thermal relay NO
	bOverload	: BOOL;
END_VAR

bOverload :=  piFR.In;
SUPER^();

PROPERTY IsOverload : REFERENCE to bool
GET
isOverload ref= bOverload;
END_GET
END_PROPERTY

PROPERTY ReasonError : string
GET
IF isOverload THEN 
	ReasonError := 'ThermalRelay OverLoad';
END_IF
END_GET
END_PROPERTY

PROPERTY Ref_piFR : reference to FB_DigitalInput
GET
Ref_piFR ref= piFR;
END_GET
END_PROPERTY

END_FUNCTION_BLOCK

// ---- POUs/Contactor/FB_ContactorNonFB_Flex.TcPOU
(* 
| :Description: This function block use for Contactor active by digital output,
| Use NO contact feedback(Digital Input) to just see, not affect the state control like "FB_contactorFBNO"
*)
FUNCTION_BLOCK FB_ContactorNonFB_Flex EXTENDS FB_ContactorNonFB
VAR
	piNO 		: FB_DigitalInputExt;
END_VAR

SUPER^();

METHOD MR_FirstCycle : BOOL
VAR_INPUT
	sName 							: STRING;
	sCoilModuleType					: STRING;
	sCoilPortID						: STRING;
	sNOModuleType					: STRING;
	sNOPortID						: STRING;
	tGoActiveTimeout				: TIME;
	tDelay							: TIME;
END_VAR
piNO.EnableTimeout := TRUE;
THIS^.sName := sName;								
THIS^.piNO.MR_FirstCycleEx(
	sName := CONCAT(sName,':NO'),
	sModuleType := sNOModuleType,
	sPortID	:= sNOPortID,
	bEnableTimeout := TRUE,
	tDefaultTimeout	:= tGoActiveTimeout
);
THIS^.poCoil.MR_FirstCycle(
	sName := CONCAT(sName,':Coil'),
	sModuleType := sCoilModuleType,
	sPortID := sCoilPortID
);
END_METHOD

PROPERTY Ref_piNO : reference to  FB_DigitalInput
GET
ref_piNO ref= THIS^.piNO;
END_GET
END_PROPERTY

END_FUNCTION_BLOCK

// ---- POUs/Contactor/FB_ContactorNonFB.TcPOU
FUNCTION_BLOCK FB_ContactorNonFB IMPLEMENTS I_ActivePowerNoFB
VAR
	sName 		: STRING;
	poCoil		: FB_DigitalOutput;
END_VAR

METHOD MR_PowerOFF : BOOL
VAR_INPUT
END_VAR
poCoil.Out := FALSE;
MR_PowerOFF := TRUE;
END_METHOD

METHOD MR_PowerON : BOOL
VAR_INPUT
END_VAR
poCoil.Out := TRUE;
MR_PowerON := TRUE;
END_METHOD

PROPERTY Name : STRING
GET
Name := sName;
END_GET
SET
sName := Name;
END_SET
END_PROPERTY

PROPERTY PowerOffIsCalled : bool
GET
PowerOffIsCalled := poCoil.Out=FALSE;
END_GET
END_PROPERTY

PROPERTY PowerOnIsCalled : bool
GET
PowerOnIsCalled := poCoil.Out=TRUE;
END_GET
END_PROPERTY

PROPERTY Ref_poCoil : reference to fb_digitalOutput
GET
ref_poCoil ref= poCoil;
END_GET
END_PROPERTY

END_FUNCTION_BLOCK

// ---- POUs/ContactorTherRelay/FB_ContactorNonFB_ThermalRelay.TcPOU
FUNCTION_BLOCK FB_ContactorNonFB_ThermalRelay EXTENDS FB_ContactorNonFB IMPLEMENTS I_ActivePowerNoFB
VAR
	piFR		: FB_DigitalInput;
	bOverload	: BOOL;
END_VAR

bOverload :=  piFR.In;
SUPER^();

PROPERTY IsOverload : REFERENCE to bool
GET
isOverload ref= bOverload;
END_GET
END_PROPERTY

PROPERTY Ref_piFR : reference to FB_DigitalInput
GET
Ref_piFR ref= piFR;
END_GET
END_PROPERTY

END_FUNCTION_BLOCK

// ---- POUs/Cylinder/Universal Cylinder/FB_UniversalCylinder.TcPOU
(* 
:Description: This function block is used represent basic cylinder device.
*)
FUNCTION_BLOCK ABSTRACT FB_UniversalCylinder IMPLEMENTS I_UniversalCylinder
VAR
	bFirstCycle			: BOOL := TRUE;			(* First cycle procedure bit *)
	sName				: STRING;				(*  *)
	
	(* Internal commands *)
	bInit 				: BOOL;					(* Prepare cylinder to work *)
	bGoActive 			: BOOL;					(* Move cylinder to active postion *)
	bGoHome 			: BOOL;					(* Move cylinder to home postion *)
	bRelease			: BOOL;					(* Release cylinder *)
	bReset				: BOOL;					(* Reset function block *)
	bAbort				: BOOL;					(* Deinitialize function block *)
	bSimulation			: BOOL;					(* Simulation on/off bit *)
	
	(* Cylinder state *)
	bActive				: BOOL;					(*  *)
	bBusy				: BOOL;					(*  *)	
	bError 				: BOOL;					(*  *)
	bPositionActive		: BOOL;					(*  *)
	bPositionHome		: BOOL;					(*  *)
	bPositionHold		: BOOL;					(*  *)
	eErrorID 			: E_CylinderError;		(*  *)
	eCylinderState		: E_CylinderState;		(* State machine of function block *)
	eCylinderGoHomeState : E_CylinderStateGo;
	eCylinderGoActiveState : E_CylinderStateGo;
	
	(* Sensors *)
	piActiveSensor		: FB_DigitalInputExt;	(* Active position sensor function block *)
	piHomeSensor		: FB_DigitalInputExt;	(* Home position sensor function block *)
	
	(* Timers *)
	tonGoHomeDelay		: TON;					(* Timer on delay when moving to home position *)
	tonGoActiveDelay	: TON;					(* Timer on delay when moving to active position *)
	tonMeasurementTimer	: TON;					(* Measurement of movement time *)
	tonCylinderWatchdog	: TON;					(* Movement watchdog *)
	
	(* Time parameters *)
	tDelay				: TIME := T#100MS;		(* Delay time when moving to any position *)
	tMeasurement		: TIME := T#60S;		(* Time of movement measurement *)

	tMoveActive			: TIME;					(* Time of last movement to active postion *)
	tMoveHome			: TIME;					(* Time of last movement to home position *)
END_VAR

(* Initial assignaments *)
IF bFirstCycle THEN
	bFirstCycle := FALSE;
	
	piHomeSensor.EnableTimeout := TRUE;
	piActiveSensor.EnableTimeout := TRUE;
END_IF

(* Simulation enabled*)
IF bSimulation THEN
	piHomeSensor.EnableForce := TRUE;
	piActiveSensor.EnableForce := TRUE;
	
	M_SimulationLogic();
ELSE
	piHomeSensor.MR_ResetForceValue();
	piActiveSensor.MR_ResetForceValue();
	piHomeSensor.EnableForce := FALSE;
	piActiveSensor.EnableForce := FALSE;
END_IF

(* Time  measurement - to active position *)
IF piActiveSensor.RisingTrigger AND eCylinderState = CYLINDER_GO_ACTIVE THEN
	tMoveActive := tonMeasurementTimer.ET;
END_IF

(* Time measurement - to home position *)
IF piHomeSensor.RisingTrigger AND eCylinderState = CYLINDER_GO_HOME THEN
	tMoveHome := tonMeasurementTimer.ET;
END_IF

(*  *)
tonMeasurementTimer(	IN := tonCylinderWatchdog.IN,
						PT := tMeasurement);

(* State machine - old *)
StateMachine();

(* Update status flags *)
bActive := eCylinderState >= CYLINDER_IDLE OR eCylinderState = CYLINDER_ABORTING ;
//bBusy := eCylinderState > CYLINDER_IDLE;
bError := piHomeSensor.ErrorTimedout OR piActiveSensor.ErrorTimedout;

(* Error handling *)
IF piHomeSensor.ErrorTimedout THEN
	eErrorID := CYLINDER_ERROR_MOVE_HOME_TIMED_OUT;
	fbMachineLogger.MR_AddLogs(FUN_MergeStrings5(sName,' : Error occured (error ID: ', 'move home timed out', ')', ''));

ELSIF piActiveSensor.ErrorTimedout THEN
	eErrorID := CYLINDER_ERROR_MOVE_ACTIVE_TIMED_OUT;
	fbMachineLogger.MR_AddLogs(FUN_MergeStrings5(sName,' : Error occured (error ID: ', 'move active timed out', ')', ''));

ELSE
	eErrorID := CYLINDER_ERROR_OK;
	
END_IF

(* Position flag update *)
bPositionActive := piActiveSensor.In;
bPositionHome := piHomeSensor.In;

(* State machine *)
//StateMachine();

(* Run sensors instances *)
piHomeSensor();
piActiveSensor();

PROPERTY Active : REFERENCE TO BOOL
GET
Active REF= bActive;
END_GET
END_PROPERTY

PROPERTY ActiveTimeout : TIME
GET
ActiveTimeout := piActiveSensor.Timeout;
END_GET
SET
piActiveSensor.Timeout := ActiveTimeout;
END_SET
END_PROPERTY

PROPERTY Busy : REFERENCE TO BOOL
GET
Busy REF= bBusy;
END_GET
END_PROPERTY

PROPERTY Delay : TIME
GET
Delay := tDelay;
END_GET
SET
tDelay := Delay;
END_SET
END_PROPERTY

PROPERTY Error : REFERENCE TO BOOL
GET
Error REF= bError;
END_GET
END_PROPERTY

PROPERTY ErrorID : REFERENCE TO E_CylinderError
GET
ErrorID REF= eErrorID;
END_GET
END_PROPERTY

PROPERTY HomeTimeout : TIME
GET
HomeTimeout := piHomeSensor.Timeout;
END_GET
SET
piHomeSensor.Timeout := HomeTimeout;
END_SET
END_PROPERTY

METHOD PROTECTED ABSTRACT M_SimulationLogic
VAR_INPUT
END_VAR
END_METHOD

PROPERTY MoveActiveTime : REFERENCE TO TIME
GET
MoveActiveTime REF= tMoveActive;
END_GET
END_PROPERTY

PROPERTY MoveHomeTime : REFERENCE TO TIME
GET
MoveHomeTime REF= tMoveHome;
END_GET
END_PROPERTY

METHOD MR_Abort : BOOL
VAR_INPUT
END_VAR
IF eCylinderState >= CYLINDER_IDLE THEN
	bBusy := TRUE;
	bAbort := TRUE;
	MR_Abort := FALSE;
	eCylinderState := CYLINDER_ABORTING;
	fbMachineLogger.MR_AddLogs(CONCAT(sName,' : abort requested'));	
	
ELSIF eCylinderState = CYLINDER_UNINITIALIZED THEN
	bAbort := FALSE;
	MR_Abort := TRUE;
	fbMachineLogger.MR_AddLogs(CONCAT(sName,' : abort done'));	
	
END_IF
END_METHOD

METHOD MR_FirstCycle : BOOL
VAR_INPUT
	sName 							: STRING;
	sHomeSensorModuleType			: STRING;
	sHomeSensorPortID				: STRING;
	sActiveSensorModuleType			: STRING;
	sActiveSensorPortID				: STRING;
	tGoHomeTimeout					: TIME;
	tGoActiveTimeout				: TIME;
	tDelay							: TIME;
END_VAR
THIS^.sName := sName;								
THIS^.tDelay := tDelay;

THIS^.piHomeSensor.MR_FirstCycleEx( sName			:= CONCAT(sName,':Home_Sensor'),
									sModuleType 	:= sHomeSensorModuleType,
									sPortID			:= sHomeSensorPortID,
									bEnableTimeout	:= TRUE,
									tDefaultTimeout	:= tGoHomeTimeout);
									
THIS^.piActiveSensor.MR_FirstCycleEx( 	sName			:= CONCAT(sName,':Active_Sensor'),
										sModuleType 	:= sActiveSensorModuleType,
										sPortID			:= sActiveSensorPortID,
										bEnableTimeout	:= TRUE,
										tDefaultTimeout	:= tGoActiveTimeout);
END_METHOD

METHOD MR_GoActive : BOOL
IF eCylinderState = CYLINDER_IDLE AND NOT piActiveSensor.In THEN
	bBusy := TRUE;
	bGoActive := TRUE;
	MR_GoActive := FALSE;
	eCylinderState := CYLINDER_GO_ACTIVE;
	eCylinderGoActiveState := CYLINDER_MOVE_START_TRACKING;
	fbMachineLogger.MR_AddLogs(CONCAT(sName,' : active position requested'));	
	
	
ELSIF eCylinderState = CYLINDER_GO_ACTIVE_DONE THEN
	bGoActive := FALSE;
	MR_GoActive := TRUE;
	fbMachineLogger.MR_AddLogs(CONCAT(sName,' : active position done'));		
	
END_IF
END_METHOD

METHOD MR_GoHome : BOOL
IF eCylinderState = CYLINDER_IDLE AND NOT piHomeSensor.In THEN
	bBusy := TRUE;
	bGoHome := TRUE;
	MR_GoHome := FALSE;
	eCylinderState := CYLINDER_GO_HOME;
	eCylinderGoHomeState := CYLINDER_MOVE_START_TRACKING;
	fbMachineLogger.MR_AddLogs(CONCAT(sName,' : home position requested'));	
	
ELSIF eCylinderState = CYLINDER_GO_HOME_DONE THEN
	bGoHome := FALSE;
	MR_GoHome := TRUE;
	fbMachineLogger.MR_AddLogs(CONCAT(sName,' : home position done'));	
	
END_IF
END_METHOD

METHOD MR_Init : BOOL
IF eCylinderState = CYLINDER_UNINITIALIZED THEN
	bBusy := TRUE;
	bInit := TRUE;
	MR_Init := FALSE;
	eCylinderState := CYLINDER_INITIALIZING;
	fbMachineLogger.MR_AddLogs(CONCAT(sName,' : initialization requested'));	
	
ELSIF eCylinderState = CYLINDER_IDLE THEN
	bInit := FALSE;
	MR_Init := TRUE;
	fbMachineLogger.MR_AddLogs(CONCAT(sName,' : initialization done'));	
	
END_IF
END_METHOD

METHOD MR_Release : BOOL
IF eCylinderState = CYLINDER_IDLE AND bPositionHold THEN
	bBusy := TRUE;
	bRelease := TRUE;
	MR_Release := FALSE;
	eCylinderState := CYLINDER_RELEASE;
	fbMachineLogger.MR_AddLogs(CONCAT(sName,' : release requested'));	
	
ELSIF eCylinderState = CYLINDER_RELEASE_DONE THEN	
	bRelease := FALSE;
	MR_Release := TRUE;
	fbMachineLogger.MR_AddLogs(CONCAT(sName,' : release done'));
	
END_IF
END_METHOD

METHOD MR_Reset : BOOL
IF eCylinderState >= CYLINDER_IDLE AND bError THEN
	bBusy := TRUE;
	bReset := TRUE;
	MR_Reset := FALSE;
	eCylinderState := CYLINDER_RESET;
	fbMachineLogger.MR_AddLogs(CONCAT(sName,' : reset requested'));	
	
ELSIF eCylinderState = CYLINDER_RESET_DONE THEN
	bReset := FALSE;
	MR_Reset := TRUE;
	fbMachineLogger.MR_AddLogs(CONCAT(sName,' : reset done'));		
	
END_IF
END_METHOD

METHOD PROTECTED  MS_Aborting
piHomeSensor.MR_Abort();
piActiveSensor.MR_Abort();

IF NOT piHomeSensor.Active AND NOT piActiveSensor.Active THEN
	//bBusy := FALSE;
	eCylinderState := CYLINDER_UNINITIALIZED;	
END_IF
END_METHOD

METHOD PROTECTED ABSTRACT MS_GoActive
END_METHOD

METHOD PROTECTED MS_GoActiveDone
IF NOT bGoActive THEN
	bBusy := FALSE;
	eCylinderState := CYLINDER_IDLE;
END_IF
END_METHOD

METHOD PROTECTED ABSTRACT MS_GoHome
END_METHOD

METHOD PROTECTED MS_GoHomeDone
IF NOT bGoHome THEN
	bBusy := FALSE;
	eCylinderState := CYLINDER_IDLE;
END_IF
END_METHOD

METHOD PROTECTED MS_Idle
;
END_METHOD

METHOD PROTECTED MS_Initializing
piHomeSensor.MR_Init();
piActiveSensor.MR_Init();

piHomeSensor.EnableTimeout := TRUE;
piActiveSensor.EnableTimeout := TRUE;

IF piHomeSensor.Active AND piActiveSensor.Active THEN
	eCylinderState := CYLINDER_READY_INITIALIZED;
END_IF
END_METHOD

METHOD PROTECTED MS_ReadyInitialized
VAR_INPUT
END_VAR
bBusy := FALSE;
eCylinderState := CYLINDER_IDLE;
END_METHOD

METHOD PROTECTED ABSTRACT MS_Release
END_METHOD

METHOD PROTECTED MS_ReleaseDone
IF NOT bRelease THEN
	bBusy := FALSE;
	eCylinderState := CYLINDER_IDLE;
END_IF
END_METHOD

METHOD PROTECTED MS_Reset
VAR_INPUT
END_VAR
bInit 		:= FALSE;
bGoActive 	:= FALSE;
bGoHome 	:= FALSE;
bRelease	:= FALSE;
bAbort		:= FALSE;

tonGoHomeDelay(IN := FALSE);
tonGoActiveDelay(IN := FALSE);
tonMeasurementTimer(IN:= FALSE);

piHomeSensor.MR_Reset();
piActiveSensor.MR_Reset();

IF NOT piHomeSensor.ErrorTimedout AND NOT piActiveSensor.ErrorTimedout THEN
	eCylinderState := CYLINDER_RESET_DONE;
END_IF
END_METHOD

METHOD PROTECTED MS_ResetDone
VAR_INPUT
END_VAR
IF NOT bReset THEN
	bBusy := FALSE;
	eCylinderState := CYLINDER_IDLE;
END_IF
END_METHOD

METHOD PROTECTED MS_Uninitialized
bError := FALSE;
bBusy := FALSE;

piHomeSensor.EnableForce := FALSE;
piActiveSensor.EnableForce := FALSE;

piHomeSensor.EnableTimeout := FALSE;
piActiveSensor.EnableTimeout := FALSE;

bInit 		:= FALSE;
bGoActive 	:= FALSE;
bGoHome 	:= FALSE;
bRelease	:= FALSE;
bReset		:= FALSE;
bAbort		:= FALSE;

tonGoHomeDelay(IN := FALSE);
tonGoActiveDelay(IN := FALSE);
tonMeasurementTimer(IN:= FALSE);
END_METHOD

PROPERTY Name : STRING
GET
Name := sName;
END_GET
SET
sName := Name;
END_SET
END_PROPERTY

PROPERTY PositionActive : REFERENCE TO BOOL
GET
PositionActive REF= bPositionActive;
END_GET
END_PROPERTY

PROPERTY PositionHold : REFERENCE TO BOOL
GET
PositionHold REF= bPositionHold;
END_GET
END_PROPERTY

PROPERTY PositionHome : REFERENCE TO BOOL
GET
PositionHome REF= bPositionHome;
END_GET
END_PROPERTY

PROPERTY ref_piActiveSensor : REFERENCE TO FB_DigitalInputExt
GET
ref_piActiveSensor REF= piActiveSensor;
END_GET
END_PROPERTY

PROPERTY ref_piHomeSensor : REFERENCE TO FB_DigitalInputExt
GET
ref_piHomeSensor REF= piHomeSensor;
END_GET
END_PROPERTY

PROPERTY Simulation : BOOL
GET
Simulation := bSimulation;
END_GET
SET
bSimulation := Simulation;
END_SET
END_PROPERTY

PROPERTY State : REFERENCE TO E_CylinderState
GET
State REF= eCylinderState;
END_GET
END_PROPERTY

METHOD PROTECTED StateMachine
CASE eCylinderState OF
	CYLINDER_UNINITIALIZED:
		MS_Uninitialized();
		
	CYLINDER_INITIALIZING:
		MS_Initializing();
	
	CYLINDER_READY_INITIALIZED:
		MS_ReadyInitialized();
		
	CYLINDER_IDLE:
		MS_Idle();
		
	CYLINDER_GO_HOME:
		MS_GoHome();
		
	CYLINDER_GO_HOME_DONE:
		MS_GoHomeDone();
		
	CYLINDER_GO_ACTIVE:
		MS_GoActive();
		
	CYLINDER_GO_ACTIVE_DONE:
		MS_GoActiveDone();
		
	CYLINDER_RELEASE:
		MS_Release();
		
	CYLINDER_RELEASE_DONE:
		MS_ReleaseDone();
		
	CYLINDER_RESET:
		MS_Reset();
		
	CYLINDER_RESET_DONE:
		MS_ResetDone();
		
	CYLINDER_ABORTING:
		MS_Aborting();
		
END_CASE
END_METHOD

END_FUNCTION_BLOCK

// ---- POUs/Digital Devices/Lamp Indicator/FB_Lamp.TcPOU
(* 
:Description: 
*)
FUNCTION_BLOCK FB_Lamp EXTENDS FB_DigitalDevice IMPLEMENTS I_Lamp
VAR
	bFirstCycle : BOOL := TRUE;
	
	poLamp				: FB_DigitalOutput;		(*  *)
	eLampState			: E_LampState;			(*  *)
	tonBlinkingTimer	: TON;					(*  *)
	tBlinkTime			: TIME;					(*  *)
	In: INT;
END_VAR

IF bFirstCycle THEN
	bFirstCycle := FALSE;
	poLamp.MR_FirstCycle(CONCAT('Digital output of: ',sName),sModuleType,sPortID);
END_IF

(*  *)
tonBlinkingTimer(	IN := (eLampState = LAMP_BLINKING_ON OR 
					eLampState = LAMP_BLINKING_OFF) AND NOT tonBlinkingTimer.Q,
					PT := tBlinkTime);

(*  *)
StateMachine();

(* *)
poLamp.Out := (eLampState = LAMP_ON OR eLampState = LAMP_BLINKING_ON);

METHOD MR_LampBlink : BOOL
VAR_INPUT
	tBlinkTime : TIME;
END_VAR
THIS^.tBlinkTime := tBlinkTime;

IF eLampState = LAMP_OFF THEN
	eLampState := LAMP_BLINKING_ON;
	
ELSIF eLampState = LAMP_ON THEN
	eLampState := LAMP_BLINKING_OFF;
	
END_IF

MR_LampBlink := TRUE;
END_METHOD

METHOD MR_LampOff : BOOL
eLampState := LAMP_OFF;
MR_LampOff := TRUE;
END_METHOD

METHOD MR_LampOn : BOOL
eLampState := LAMP_ON;
MR_LampOn := TRUE;
END_METHOD

METHOD PROTECTED MS_LampBlinkingOff
VAR_INPUT
END_VAR
IF tonBlinkingTimer.Q THEN
	eLampState := LAMP_BLINKING_ON;
END_IF
END_METHOD

METHOD PROTECTED MS_LampBlinkingOn
VAR_INPUT
END_VAR
IF tonBlinkingTimer.Q THEN
	eLampState := LAMP_BLINKING_OFF;
END_IF
END_METHOD

METHOD PROTECTED MS_LampOff
VAR_INPUT
END_VAR
;
END_METHOD

METHOD PROTECTED MS_LampOn
VAR_INPUT
END_VAR
;
END_METHOD

METHOD PROTECTED StateMachine
VAR_INPUT
END_VAR
(*  *)
CASE eLampState OF
	LAMP_OFF:
		MS_LampOff();
		
	LAMP_ON:
		MS_LampOn();
		
	LAMP_BLINKING_ON:
		MS_LampBlinkingOn();
		
	LAMP_BLINKING_OFF:
		MS_LampBlinkingOff();
	
END_CASE
END_METHOD

PROPERTY Status : REFERENCE TO E_LampState
GET
Status REF= eLampState;
END_GET
END_PROPERTY

END_FUNCTION_BLOCK

// ---- POUs/Tank0FB/FB_SingleTankSV1Ext.TcPOU
FUNCTION_BLOCK FB_SingleTankSV1Ext EXTENDS FB_SingleTankSV1
VAR
	sNameTask : STRING;
	bBusyTask : BOOL;
END_VAR

SUPER^();

PROPERTY BusyTask : BOOL
GET
BusyTask := bBusyTask;
END_GET
END_PROPERTY

METHOD RegisterTask : BOOL
VAR_INPUT
	sTask : STRING;
END_VAR
IF NOT bBusyTask THEN
	sNameTask := sTask;
	bBusyTask := true;
	RegisterTask := TRUE;
ELSE
	RegisterTask := FALSE;
END_IF
END_METHOD

PROPERTY TaskRegistered : string
GET
TaskRegistered := sNameTask;
END_GET
END_PROPERTY

METHOD UnRegisterTask : BOOL
VAR_INPUT
END_VAR
bBusyTask := FALSE;
sNameTask := '';
UnRegisterTask := true;
END_METHOD

END_FUNCTION_BLOCK

// ---- POUs/Tank0FB/FB_SingleTankSV1.TcPOU
(* Single tank with LimitSwitchLow (piLsLow) and LimitSwitchHigh (piLsHigh)
| using this function when it have INDEPENDENT Measure weight
*)
FUNCTION_BLOCK FB_SingleTankSV1 EXTENDS FB_SingleTankS
VAR
	bAllowInMaterial : BOOL;
	bAllowOutMaterial : BOOL;
	lrLimitMinWeight : LREAL;
	lrLimitMaxWeight : LREAL;
	lrWeightWithdraw : LREAL; 		// weight withdraw Request
	lrWeightBeforeWD : LREAL;
	lrWeightWithdrawN : LREAL;
	lrWeight : LREAL;
	eState : E_TankState;
	iFill : I_TankFill;				// the components that action for fill materials.
	
	rTrigExecute : R_TRIG;
	bExecute : BOOL;//Execute with draw
	bFillError : BOOL;
	bError : BOOL;
	bWithDrawDone : BOOL;
	tonWithDrawStable : TON;
	tTimeWithDrawStable : TIME := T#3S;
	bEnoughWithdraw : BOOL;
END_VAR

SUPER^();
rTrigExecute(CLK := bExecute);
bAllowOutMaterial := (lrWeight > lrLimitMinWeight);
bAllowInMaterial := (lrWeight < lrLimitMaxWeight);
lrWeightWithdrawN := lrWeightBeforeWD-lrWeight;
tonWithDrawStable(IN := eState=TANK_WITHDRAWING_DONE, PT := tTimeWithDrawStable);
CASE eState OF
	TANK_IDLE:
		;// WAIT FOR CMD
	TANK_STOP:
		MS_Stop();
		
	TANK_WITHDRAWING:
		MS_Withdraw();
		
	TANK_WITHDRAWING_DONE:
		Ms_WithDrawDone();
		
	TANK_FILLING:
		MS_Filling();
END_CASE

PROPERTY AllowIn : Reference to bool
GET
AllowIn ref= bAllowInMaterial;
END_GET
END_PROPERTY

(*
| Check the minimum condition  (lrWeight > lrLimitMinWeight
								AND piLslow.In;)
*)
PROPERTY AllowOut : REFERENCE TO BOOL
GET
AllowOut ref= bAllowOutMaterial;
END_GET
END_PROPERTY

METHOD AssignIfill : BOOL
VAR_INPUT
	iFill : I_TankFill;
END_VAR
THIS^.iFill := iFill;
END_METHOD

METHOD CheckEnoughWithDraw : BOOL
VAR_INPUT
	lrWeightWd : LREAL;
END_VAR
IF 	lrWeight > (lrWeightWd + lrLimitMinWeight) THEN
	bEnoughWithdraw := TRUE;
ELSE
	bEnoughWithdraw := FALSE;
END_IF
CheckEnoughWithDraw := bEnoughWithdraw;
END_METHOD

PROPERTY Error : reference to Bool
GET
Error ref= bError;
END_GET
END_PROPERTY

PROPERTY LimitMaxWeight : LREAL
GET
LimitMaxWeight := lrLimitMaxWeight;
END_GET
SET
lrLimitMaxWeight := LimitMaxWeight;
END_SET
END_PROPERTY

PROPERTY LimitMinWeight : LREAL
GET
LimitMinWeight := lrLimitMinWeight;
END_GET
SET
lrLimitMinWeight := LimitMinWeight;
END_SET
END_PROPERTY

METHOD MR_Filling : BOOL
VAR_INPUT
END_VAR
IF eState=TANK_IDLE 
	AND bAllowInMaterial
THEN
	eState := TANK_FILLING;
END_IF
END_METHOD

METHOD MR_Reset : BOOL
VAR_INPUT
END_VAR
bError := FALSE;
bWithDrawDone := FALSE;
MR_Reset := TRUE;
END_METHOD

METHOD MR_Stop : BOOL
VAR_INPUT
END_VAR
eState := TANK_STOP;
END_METHOD

(*	
	please call bExecute := false and then call bExecute := true for begin withdraw 
	if withdrawing => still withdraw
	else
		if not stop => MR_Stop before withdraw
*)
METHOD MR_WithDraw : BOOL
VAR_INPUT
	lrWeightWd : LREAL;
	bExecute : BOOL;
END_VAR
THIS^.bExecute := bExecute;
IF rTrigExecute.Q
	AND eState=TANK_IDLE 
	AND lrWeight > (lrWeightWd + lrLimitMinWeight) // Check enough weight
	AND bAllowOutMaterial
THEN
	eState := TANK_WITHDRAWING;
	lrWeightWithdraw := lrWeightWd;
	lrWeightBeforeWD := lrWeight;
END_IF
IF bExecute= FALSE THEN
	bWithDrawDone := FALSE;
END_IF
END_METHOD

METHOD PROTECTED MS_Filling
VAR_INPUT
END_VAR
IF bAllowInMaterial THEN
	iFill.Open();
ELSE
	iFill.Close();
	bError := TRUE;
	eState := TANK_STOP;
END_IF
END_METHOD

METHOD PROTECTED MS_Stop
VAR_INPUT
END_VAR
poCylinderCoil.Out := FALSE;
iFill.Close();
bExecute := FALSE;
eState := TANK_IDLE;
END_METHOD

METHOD PROTECTED MS_Withdraw
VAR_INPUT
END_VAR
poCylinderCoil.Out := TRUE;
IF lrWeightWithdrawN > lrWeightWithdraw THEN
	eState := TANK_WITHDRAWING_DONE;
END_IF
IF NOT bAllowOutMaterial THEN
	bError := TRUE;
END_IF
END_METHOD

METHOD PROTECTED MS_WithDrawDone : BOOL
VAR_INPUT
END_VAR
poCylinderCoil.Out := FALSE;
IF tonWithDrawStable.Q THEN
	bWithDrawDone := TRUE;
	eState := TANK_IDLE;
END_IF
END_METHOD

PROPERTY Ref_iFill : Reference to I_TankFill
GET
Ref_iFill ref= iFill;
END_GET
END_PROPERTY

PROPERTY TimeWithDrawStable : Time
GET
TimeWithDrawStable := tTimeWithDrawStable;
END_GET
SET
tTimeWithDrawStable := TimeWithDrawStable;
END_SET
END_PROPERTY

PROPERTY Weight : lreal
GET
Weight := lrWeight;
END_GET
SET
Weight := lrWeight;
END_SET
END_PROPERTY

PROPERTY WeightWithdraw : lreal
GET
WeightWithdraw := lrWeightWithdraw;
END_GET
SET
lrWeightWithdraw := WeightWithdraw;
END_SET
END_PROPERTY

PROPERTY WeightWithDrawN : lreal
GET
WeightWithDrawN := lrWeightWithdrawN;
END_GET
END_PROPERTY

PROPERTY WithDrawDone : Bool
GET
WithDrawDone := bWithDrawDone;
END_GET
END_PROPERTY

END_FUNCTION_BLOCK

// ---- POUs/Tank0FB/FB_SingleTankS.TcPOU
FUNCTION_BLOCK FB_SingleTankS
VAR
	sName : STRING;
	sWeightUnit : STRING := 'Kg'; // Kg
	poCylinderCoil : FB_DigitalOutput;
END_VAR

PROPERTY Name : String
GET
Name := sName;
END_GET
SET
sName := Name;
END_SET
END_PROPERTY

PROPERTY Ref_poCylinderCoil : REFERENCE TO FB_DigitalOutput
GET
Ref_poCylinderCoil ref= poCylinderCoil;
END_GET
END_PROPERTY

PROPERTY WeightUnit : string
GET
WeightUnit := sWeightUnit;
END_GET
SET
sWeightUnit := WeightUnit;
END_SET
END_PROPERTY

END_FUNCTION_BLOCK

// ---- POUs/TankFB/FB_SingleTankV0.TcPOU
(* Single tank with LimitSwitchLow (piLsLow) and LimitSwitchHigh (piLsHigh)
| using this function when have to DEPENDENT Measure weight
*)
FUNCTION_BLOCK FB_SingleTankV0 EXTENDS FB_SingleTank
VAR
	bAllowInMaterial : BOOL;
	bAllowOutMaterial : BOOL;
	tonRemainOffLsLow	: TON;
	tRemainOffLsLow	: TIME := T#1S;
	tonRemainLsHigh	: TON;
	tRemainLsHigh	: TIME := T#1S;	
END_VAR

tonRemainOffLsLow(
	IN := NOT piLslow.In,
	PT := tRemainOffLsLow,
);
bAllowOutMaterial := NOT tonRemainOffLsLow.Q;

tonRemainLsHigh(
	IN := piLsHigh.In,
	PT := tRemainLsHigh,
);
bAllowInMaterial := NOT tonRemainLsHigh.Q;
SUPER^();

PROPERTY AllowIn : Reference to bool
GET
AllowIn ref= bAllowInMaterial;
END_GET
END_PROPERTY

(*
| Check the minimum condition  (lrWeight > lrLimitMinWeight
								AND piLslow.In;)
*)
PROPERTY AllowOut : REFERENCE TO BOOL
GET
AllowOut ref= bAllowOutMaterial;
END_GET
END_PROPERTY

PROPERTY TimeRemainLsHigh : Time
GET
TimeRemainLsHigh := tRemainLsHigh;
END_GET
SET
tRemainLsHigh := TimeRemainLsHigh;
END_SET
END_PROPERTY

PROPERTY TimeRemainOffLsLow : Time
GET
TimeRemainOffLsLow := tRemainOffLsLow;
END_GET
SET
tRemainOffLsLow := TimeRemainOffLsLow;
END_SET
END_PROPERTY

END_FUNCTION_BLOCK

// ---- POUs/TankFB/FB_SingleTankV1.TcPOU
(* Single tank with LimitSwitchLow (piLsLow) and LimitSwitchHigh (piLsHigh)
| using this function when it have INDEPENDENT Measure weight
*)
FUNCTION_BLOCK FB_SingleTankV1 EXTENDS FB_SingleTank
VAR
	bAllowInMaterial : BOOL;
	bAllowOutMaterial : BOOL;
	lrLimitMinWeight : LREAL;
	lrLimitMaxWeight : LREAL;
	lrWeightWithdraw : LREAL; 		// weight withdraw Request
	lrWeightBeforeWD : LREAL;
	lrWeightWithdrawN : LREAL;
	lrWeight : LREAL;
	eState : E_TankState;
	iFill : I_TankFill;				// the components that action for fill materials.
	
	tonRemainOffLsLow	: TON;
	tRemainOffLsLow	: TIME := T#1S;
	tonRemainLsHigh	: TON;
	tRemainLsHigh	: TIME := T#1S;	
	rTrigExecute : R_TRIG;
	bExecute : BOOL;//Execute with draw
	bFillError : BOOL;
	bError : BOOL;
END_VAR

SUPER^();
rTrigExecute(CLK := bExecute);
tonRemainOffLsLow(
	IN := NOT piLslow.In,
	PT := tRemainOffLsLow,
);
bAllowOutMaterial := (lrWeight > lrLimitMinWeight) AND NOT tonRemainOffLsLow.Q;

tonRemainLsHigh(
	IN := piLsHigh.In,
	PT := tRemainLsHigh,
);
bAllowInMaterial := (lrWeight < lrLimitMaxWeight) AND NOT tonRemainLsHigh.Q;
lrWeightWithdrawN := lrWeightBeforeWD-lrWeight;

CASE eState OF
	TANK_STOP:
		MS_Stop();
		
	TANK_WITHDRAWING:
		MS_Withdraw();
		
	TANK_FILLING:
		MS_Filling();
END_CASE

PROPERTY AllowIn : Reference to bool
GET
AllowIn ref= bAllowInMaterial;
END_GET
END_PROPERTY

(*
| Check the minimum condition  (lrWeight > lrLimitMinWeight
								AND piLslow.In;)
*)
PROPERTY AllowOut : REFERENCE TO BOOL
GET
AllowOut ref= bAllowOutMaterial;
END_GET
END_PROPERTY

METHOD AssignIfill : BOOL
VAR_INPUT
	iFill : I_TankFill;
END_VAR
THIS^.iFill := iFill;
END_METHOD

PROPERTY Error : reference to Bool
GET
Error ref= bError;
END_GET
END_PROPERTY

PROPERTY LimitMaxWeight : LREAL
GET
LimitMaxWeight := lrLimitMaxWeight;
END_GET
SET
lrLimitMaxWeight := LimitMaxWeight;
END_SET
END_PROPERTY

PROPERTY LimitMinWeight : LREAL
GET
LimitMinWeight := lrLimitMinWeight;
END_GET
SET
lrLimitMinWeight := LimitMinWeight;
END_SET
END_PROPERTY

METHOD MR_Filling : BOOL
VAR_INPUT
END_VAR
IF eState=TANK_STOP 
	AND bAllowInMaterial
THEN
	eState := TANK_FILLING;
END_IF
END_METHOD

METHOD MR_Reset : BOOL
VAR_INPUT
END_VAR
bError := FALSE;
MR_Reset := TRUE;
END_METHOD

METHOD MR_Stop : BOOL
VAR_INPUT
END_VAR
eState := TANK_STOP;
END_METHOD

(*	if withdrawing => still withdraw
	else
		if not stop => MR_Stop before withdraw
*)
METHOD MR_WithDraw : BOOL
VAR_INPUT
	lrWeightWd : LREAL;
	bExecute : BOOL;
END_VAR
THIS^.bExecute := bExecute;
IF rTrigExecute.Q
	AND eState=TANK_STOP 
	AND lrWeight > (lrWeightWd + lrLimitMinWeight) // Check enough weight
	AND bAllowOutMaterial
THEN
	eState := TANK_WITHDRAWING;
	lrWeightWithdraw := lrWeightWd;
	lrWeightBeforeWD := lrWeight;
END_IF
END_METHOD

METHOD PROTECTED MS_Filling
VAR_INPUT
END_VAR
IF bAllowInMaterial THEN
	iFill.Open();
ELSE
	iFill.Close();
	bError := TRUE;
	eState := TANK_STOP;
END_IF
END_METHOD

METHOD PROTECTED MS_Stop
VAR_INPUT
END_VAR
poCylinderCoil.Out := FALSE;
iFill.Close();
END_METHOD

METHOD PROTECTED MS_Withdraw
VAR_INPUT
END_VAR
poCylinderCoil.Out := TRUE;
IF lrWeightWithdrawN > lrWeightWithdraw THEN
	eState := TANK_STOP;
END_IF
IF NOT bAllowOutMaterial THEN
	bError := TRUE;
END_IF
END_METHOD

PROPERTY Ref_iFill : Reference to I_TankFill
GET
Ref_iFill ref= iFill;
END_GET
END_PROPERTY

PROPERTY TimeRemainLsHigh : Time
GET
TimeRemainLsHigh := tRemainLsHigh;
END_GET
SET
tRemainLsHigh := TimeRemainLsHigh;
END_SET
END_PROPERTY

PROPERTY TimeRemainOffLsLow : Time
GET
TimeRemainOffLsLow := tRemainOffLsLow;
END_GET
SET
tRemainOffLsLow := TimeRemainOffLsLow;
END_SET
END_PROPERTY

PROPERTY Weight : lreal
GET
Weight := lrWeight;
END_GET
SET
Weight := lrWeight;
END_SET
END_PROPERTY

PROPERTY WeightWithdraw : lreal
GET
WeightWithdraw := lrWeightWithdraw;
END_GET
SET
lrWeightWithdraw := WeightWithdraw;
END_SET
END_PROPERTY

END_FUNCTION_BLOCK

// ---- POUs/TankFB/FB_TankFourCompartments.TcPOU
(* FB_TankFourCompartments contain 4 SingleTank
*)
FUNCTION_BLOCK FB_TankFourCompartments
VAR
	sName : STRING;
	lrWeight : LREAL;				//Total Weight of the 4 tanks
	sWeightUnit : STRING := 'Kg'; 	// Kg
	fbTank1 : FB_SingleTankV0;
	fbTank2 : FB_SingleTankV0;
	fbTank3 : FB_SingleTankV0;
	fbTank4 : FB_SingleTankV0;
	
	bAllowInMaterial : BOOL;
	bAllowOutMaterial : BOOL;
	lrLimitMinWeight : LREAL;
	lrLimitMaxWeight : LREAL;
	lrWeightWithdraw : LREAL; 		// weight withdraw Request 
	bEnoughWithdraw : BOOL;
END_VAR

fbTank1();
fbTank2();
fbTank3();
fbTank4();
bAllowInMaterial := lrWeight < lrLimitMaxWeight;	
bAllowOutMaterial := lrWeight > lrLimitMinWeight;
bEnoughWithdraw := lrWeight > (lrWeightWithdraw + lrLimitMinWeight);

PROPERTY AllowIn : Reference to bool
GET
AllowIn ref= bAllowInMaterial;
END_GET
END_PROPERTY

(*
| Check the minimum condition  (lrWeight > lrLimitMinWeight
								AND piLslow.In;)
*)
PROPERTY AllowOut : REFERENCE TO BOOL
GET
AllowOut ref= bAllowOutMaterial;
END_GET
END_PROPERTY

(*
|Check every single tank enough weight to withdraw
|I'm not sure whether this function CLEAN ? SOLID principle
*)
PROPERTY EnoughWithdraw : reference to bool
GET
EnoughWithdraw ref= bEnoughWithdraw;
END_GET
END_PROPERTY

METHOD FirstCycle : BOOL
VAR_INPUT
	sName : STRING;
	sWeightUnit : STRING;
END_VAR
THIS^.sName := sName;
THIS^.sWeightUnit := sWeightUnit;

fbTank1.Name := CONCAT(sName, ' part 1');
fbTank1.WeightUnit := sWeightUnit;

fbTank2.Name := CONCAT(sName, ' part 2');
fbTank2.WeightUnit := sWeightUnit;

fbTank3.Name := CONCAT(sName, ' part 3');
fbTank3.WeightUnit := sWeightUnit;

fbTank4.Name := CONCAT(sName, ' part 4');
fbTank4.WeightUnit := sWeightUnit;
END_METHOD

PROPERTY LimitMaxWeight : lreal
GET
LimitMaxWeight := lrLimitMaxWeight;
END_GET
SET
lrLimitMaxWeight := LimitMaxWeight;
END_SET
END_PROPERTY

PROPERTY LimitMinWeight : lreal
GET
LimitMinWeight := lrLimitMinWeight;
END_GET
SET
lrLimitMinWeight := LimitMinWeight;
END_SET
END_PROPERTY

PROPERTY Name : String
GET
Name := sName;
END_GET
SET
sName := Name;
END_SET
END_PROPERTY

PROPERTY Ref_Tank1 : Reference to FB_SingleTankV0
GET
Ref_Tank1 ref= fbTank1;
END_GET
END_PROPERTY

PROPERTY Ref_Tank2 : Reference to FB_SingleTankV0
GET
Ref_Tank2 ref= fbTank2;
END_GET
END_PROPERTY

PROPERTY Ref_Tank3 : Reference to FB_SingleTankV0
GET
Ref_Tank3 ref= fbTank3;
END_GET
END_PROPERTY

PROPERTY Ref_Tank4 : Reference to FB_SingleTankV0
GET
Ref_Tank4 ref= fbTank4;
END_GET
END_PROPERTY

PROPERTY Weight : lreal
GET
Weight := lrWeight;
END_GET
SET
lrWeight := Weight;
END_SET
END_PROPERTY

PROPERTY WeightUnit : string
GET
WeightUnit := sWeightUnit;
END_GET
SET
sWeightUnit := WeightUnit;
END_SET
END_PROPERTY

PROPERTY WeightWithdraw : lreal
GET
WeightWithdraw := lrWeightWithdraw;
END_GET
SET
lrWeightWithdraw := WeightWithdraw;
END_SET
END_PROPERTY

END_FUNCTION_BLOCK

// ---- POUs/TankFB/Fill/FB_TankFill_2Cylinder.TcPOU
(*P&ID: 2 cylinder but Actual design 1 cylinder1*)
FUNCTION_BLOCK FB_TankFill_2Cylinder IMPLEMENTS I_TankFill
VAR
	poCylinder1 : FB_DigitalOutput;
	poCylinder2 : FB_DigitalOutput;
END_VAR

poCylinder1();
poCylinder2();

METHOD Close : BOOL
VAR_INPUT
END_VAR
poCylinder1.Out := FALSE;
poCylinder2.Out := FALSE;
END_METHOD

PROPERTY IsClose : bool
GET
IsClose := poCylinder1.Out=false;
END_GET
END_PROPERTY

PROPERTY IsOpen : bool
GET
IsOpen := poCylinder1.Out=True;
END_GET
END_PROPERTY

METHOD Open : BOOL
VAR_INPUT
END_VAR
poCylinder1.Out := TRUE;
poCylinder2.Out := TRUE;
END_METHOD

PROPERTY Ref_poCylinder1 : Reference to FB_DigitalOutput
GET
Ref_poCylinder1 ref= poCylinder1;
END_GET
END_PROPERTY

PROPERTY Ref_poCylinder2 : Reference to FB_DigitalOutput
GET
Ref_poCylinder2 ref= poCylinder2;
END_GET
END_PROPERTY

END_FUNCTION_BLOCK

// ---- POUs/TankMix/FB_Mixer0.TcPOU
(*The tank with opened lid and have a motor for mix, a cylinder for out material*)
FUNCTION_BLOCK FB_Mixer0
VAR
	poCylinderOut : FB_DigitalOutput;
	fbMotorContactor : FB_ContactorNonFB_ThermalRelay;
END_VAR

poCylinderOut();
fbMotorContactor();

METHOD Mix : BOOL
VAR_INPUT
END_VAR
fbMotorContactor.MR_PowerON();
END_METHOD

METHOD OutMaterial : BOOL
VAR_INPUT
END_VAR
poCylinderOut.Out := true;
END_METHOD

PROPERTY Ref_MotorContactor : REFERENCE TO FB_ContactorNonFB_ThermalRelay
GET
Ref_MotorContactor ref= fbMotorContactor;
END_GET
END_PROPERTY

PROPERTY Ref_poCylinderOut : reference to FB_DigitalOutput
GET
Ref_poCylinderOut ref= poCylinderOut;
END_GET
END_PROPERTY

METHOD StopAll : BOOL
VAR_INPUT
END_VAR
StopMix();
StopOutMaterial();
END_METHOD

METHOD StopMix : BOOL
VAR_INPUT
END_VAR
fbMotorContactor.MR_PowerOFF();
END_METHOD

METHOD StopOutMaterial : BOOL
VAR_INPUT
END_VAR
poCylinderOut.Out := false;
END_METHOD

END_FUNCTION_BLOCK

// ---- GlobalTextList.TcGTLO
TEXTLIST GlobalTextList
  331 = '%d'
  976 = '%s'
  2051 = '/'
  887 = 'Abort'
  424 = 'Cylinders'
  1456 = 'Digital inputs'
  1445 = 'Digital outputs'
  537 = 'Error: %d'
  244 = 'Go %s'
  371 = 'Initialize'
  1606 = 'Next'
  1146 = 'Parameters:'
  1845 = 'Position hold'
  905 = 'Position: %s'
  1825 = 'Previous'
  1083 = 'Release'
  3075 = 'Reset'
  2584 = 'Safe Inputs'
  1087 = 'Safe Outputs'
  670 = 'Safety I/O'
  1037 = 'State: %s'
END_TEXTLIST

// ---- VISUs/Pages/PageManualCylinders.TcVIS
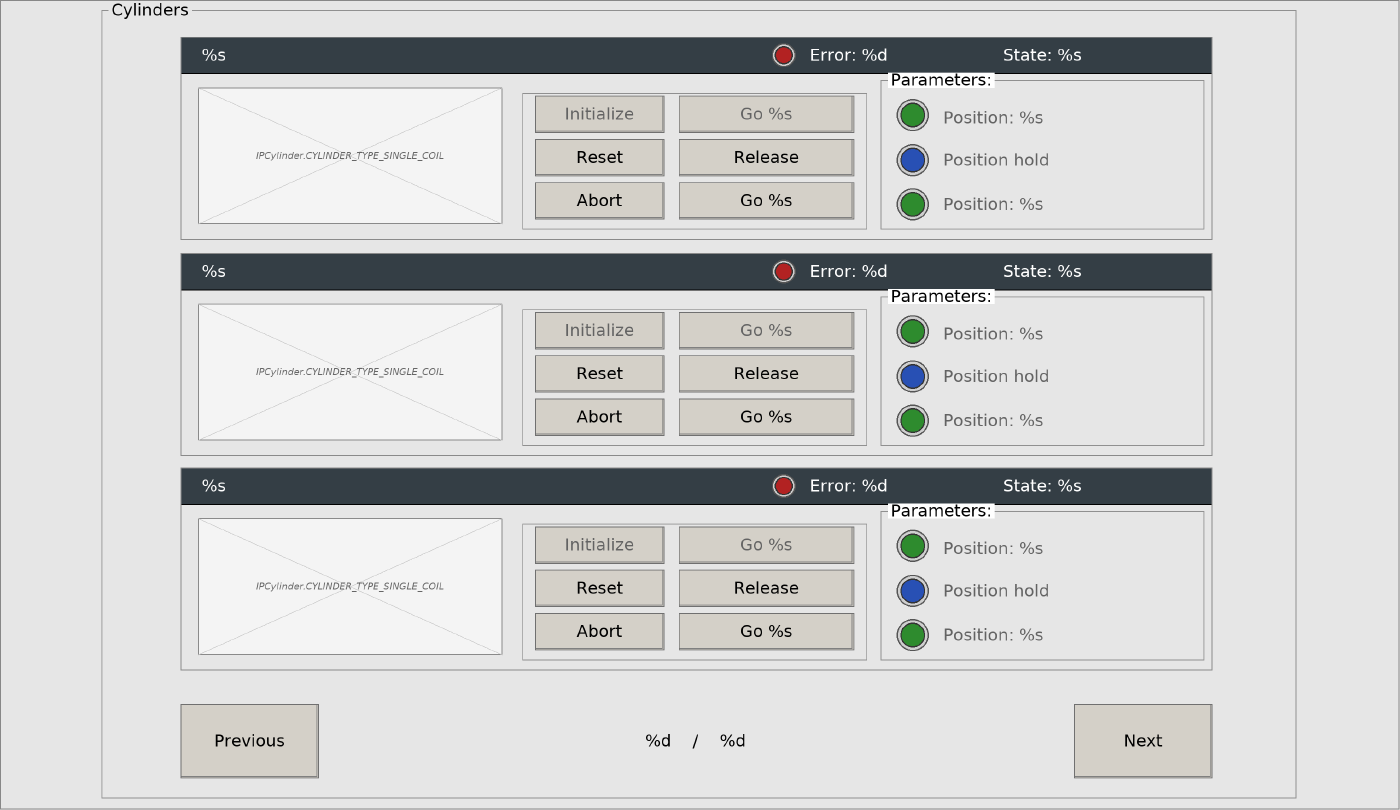
VISUALIZATION PageManualCylinders  // 1520x880
VAR_IN_OUT
	btnPrevious			: BOOL;
	btnNext				: BOOL;
	bPreviousInvisible	: BOOL;
	bNextInvisible		: BOOL;
	stCylinderEmpty		: ARRAY[1..3] OF BOOL;
	stCyliner			: ARRAY[1..3] OF ST_VisuCtrlCylinderFrame;
	iCylinderSelectedPageIndex	: USINT;
	iCylinderTotalPageIndex 	: USINT;
END_VAR
    GroupBox (110,3 1297x864), "Cylinders"
        Button (86,762 150x80), "Previous", invisible if: bPreviousInvisible
            tap btnPrevious
        Button (1056,762 150x80), "Next", invisible if: bNextInvisible
            tap btnNext
        Frame (86,37 1120x220), invisible if: stCylinderEmpty[1]
            shows SingleCylinder(stCylinder := stCyliner[1])
        Frame (86,272 1120x220), invisible if: stCylinderEmpty[2]
            shows SingleCylinder(stCylinder := stCyliner[2])
        Frame (86,505 1120x220), invisible if: stCylinderEmpty[3]
            shows SingleCylinder(stCylinder := stCyliner[3])
        Rectangle (580,777 130x50), "/"
        Rectangle (580,777 50x50), "%d", text variable: iCylinderSelectedPageIndex+1
        Rectangle (661,777 50x50), "%d", text variable: iCylinderTotalPageIndex+1
END_VISUALIZATION

// ---- VISUs/Pages/PageManualInputs.TcVIS
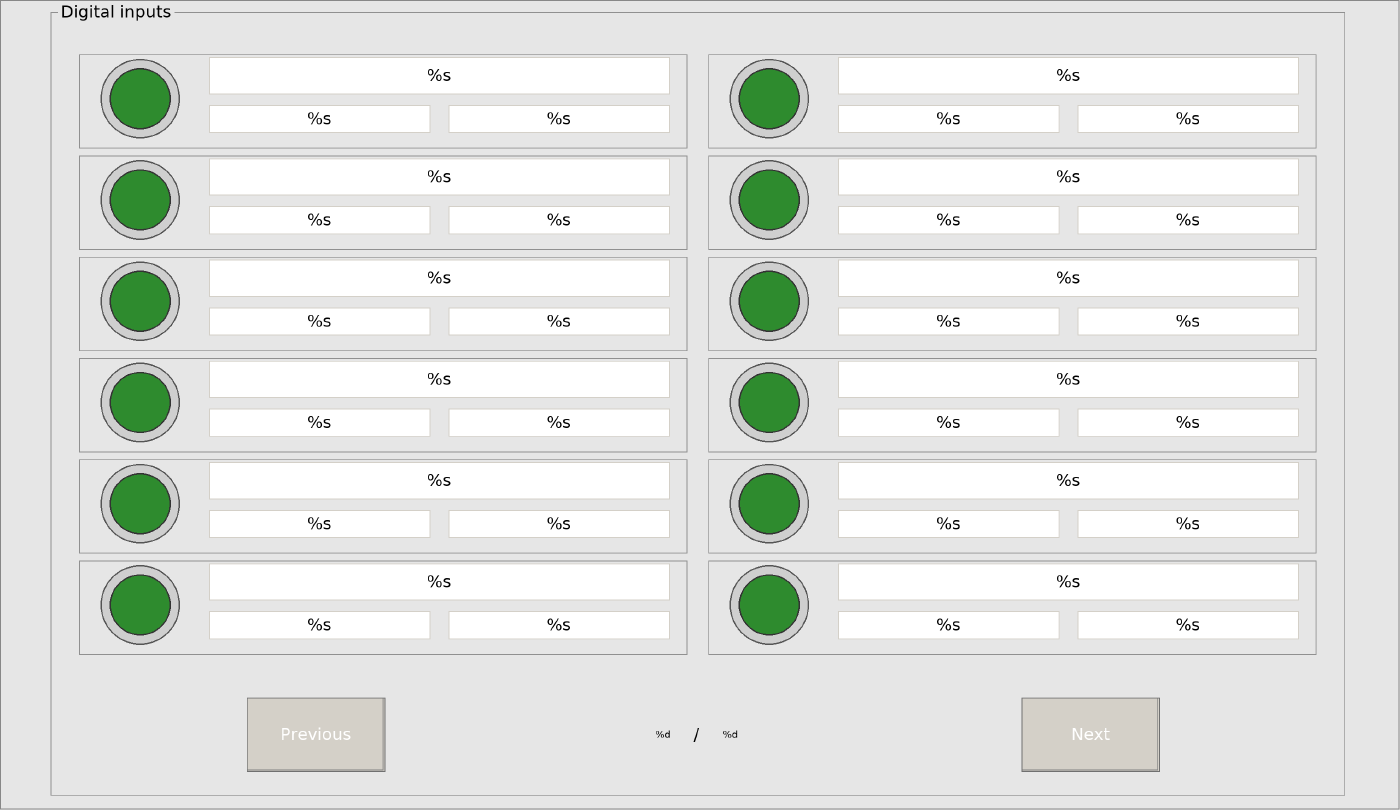
VISUALIZATION PageManualInputs  // 1520x880
VAR_IN_OUT
	btnPrevious			: BOOL;
	btnNext				: BOOL;
	
	bPreviousInvisible	: BOOL;
	bNextInvisible		: BOOL;
	
	stDigitalInputEmpty	: ARRAY[1..12] OF BOOL;
	stDigitalInputData	: ARRAY[1..12] OF ST_VisuCtrlInputFrame;
	
	iInputSelectedPageIndex		: USINT;
	iInputTotalPageIndex 		: USINT;
END_VAR
    GroupBox (55,5 1405x859), "Digital inputs"
        Rectangle (713,768 50x50), "%d", text variable: iInputTotalPageIndex+1
        Rectangle (640,768 50x50), "%d", text variable: iInputSelectedPageIndex+1
        Rectangle (636,768 130x50), "/"
        Button (213,753 150x80), "Previous", invisible if: bPreviousInvisible
            tap btnPrevious
        Button (1054,753 150x80), "Next", invisible if: bNextInvisible
            tap btnNext
        Frame (31,46 660x110), invisible if: stDigitalInputEmpty[1]
            shows SingleDigitalInput(stDigitalInput := stDigitalInputData[1])
        Frame (31,156 660x110), invisible if: stDigitalInputEmpty[2]
            shows SingleDigitalInput(stDigitalInput := stDigitalInputData[2])
        Frame (31,266 660x110), invisible if: stDigitalInputEmpty[3]
            shows SingleDigitalInput(stDigitalInput := stDigitalInputData[3])
        Frame (31,376 660x110), invisible if: stDigitalInputEmpty[4]
            shows SingleDigitalInput(stDigitalInput := stDigitalInputData[4])
        Frame (31,486 660x110), invisible if: stDigitalInputEmpty[5]
            shows SingleDigitalInput(stDigitalInput := stDigitalInputData[5])
        Frame (31,596 660x110), invisible if: stDigitalInputEmpty[6]
            shows SingleDigitalInput(stDigitalInput := stDigitalInputData[6])
        Frame (714,46 660x110), invisible if: stDigitalInputEmpty[7]
            shows SingleDigitalInput(stDigitalInput := stDigitalInputData[7])
    Frame (769,161 660x110), invisible if: stDigitalInputEmpty[8]
        shows SingleDigitalInput(stDigitalInput := stDigitalInputData[8])
    Frame (769,271 660x110), invisible if: stDigitalInputEmpty[9]
        shows SingleDigitalInput(stDigitalInput := stDigitalInputData[9])
    Frame (769,381 660x110), invisible if: stDigitalInputEmpty[10]
        shows SingleDigitalInput(stDigitalInput := stDigitalInputData[10])
    Frame (769,491 660x110), invisible if: stDigitalInputEmpty[11]
        shows SingleDigitalInput(stDigitalInput := stDigitalInputData[11])
    Frame (769,601 660x110), invisible if: stDigitalInputEmpty[12]
        shows SingleDigitalInput(stDigitalInput := stDigitalInputData[12])
END_VISUALIZATION

// ---- VISUs/Pages/PageManualOutputs.TcVIS
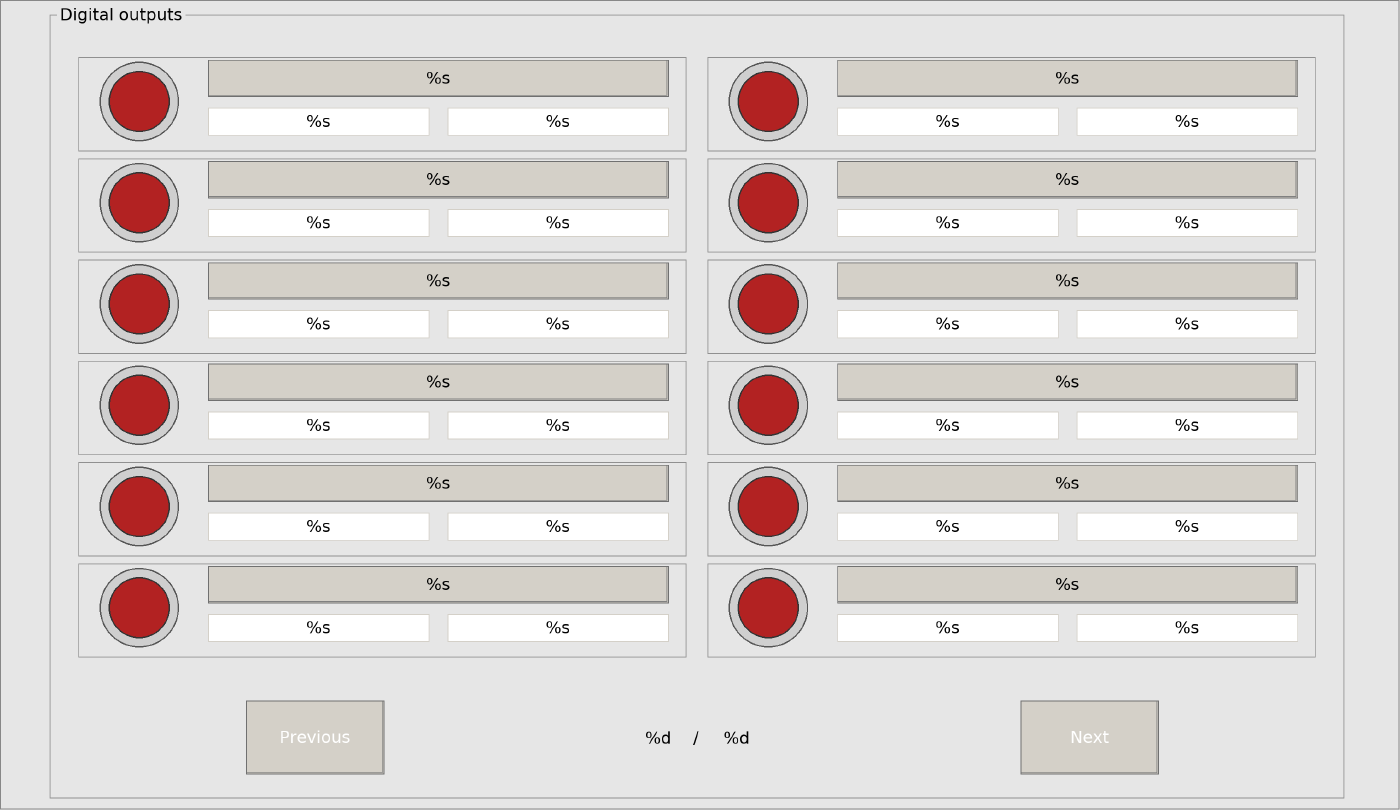
VISUALIZATION PageManualOutputs  // 1520x880
VAR_IN_OUT
	btnPrevious			: BOOL;
	btnNext				: BOOL;
	
	bPreviousInvisible	: BOOL;
	bNextInvisible		: BOOL;
	
	stDigitalOutputEmpty: ARRAY[1..12] OF BOOL;
	stDigitalOutputData	: ARRAY[1..12] OF ST_VisuCtrlOutputFrame;
	
	iOutputSelectedPageIndex	: USINT;
	iOutputTotalPageIndex 		: USINT;
END_VAR
    GroupBox (54,8 1405x859), "Digital outputs"
        Rectangle (721,769 50x50), "%d", text variable: iOutputTotalPageIndex + 1
        Rectangle (636,769 50x50), "%d", text variable: iOutputSelectedPageIndex+1
        Rectangle (636,768 131x51), "/"
        Button (213,753 150x80), "Previous", invisible if: bPreviousInvisible
            tap btnPrevious
        Button (1054,753 150x80), "Next", invisible if: bNextInvisible
            tap btnNext
        Frame (31,46 660x110), invisible if: stDigitalOutputEmpty[1]
            shows SingleDigitalOutput(stDigitalOutput := stDigitalOutputData[1])
        Frame (31,156 660x110), invisible if: stDigitalOutputEmpty[2]
            shows SingleDigitalOutput(stDigitalOutput := stDigitalOutputData[2])
        Frame (31,266 660x110), invisible if: stDigitalOutputEmpty[3]
            shows SingleDigitalOutput(stDigitalOutput := stDigitalOutputData[3])
        Frame (31,376 660x110), invisible if: stDigitalOutputEmpty[4]
            shows SingleDigitalOutput(stDigitalOutput := stDigitalOutputData[4])
        Frame (31,486 660x110), invisible if: stDigitalOutputEmpty[5]
            shows SingleDigitalOutput(stDigitalOutput := stDigitalOutputData[5])
        Frame (31,596 660x110), invisible if: stDigitalOutputEmpty[6]
            shows SingleDigitalOutput(stDigitalOutput := stDigitalOutputData[6])
        Frame (714,46 660x110), invisible if: stDigitalOutputEmpty[7]
            shows SingleDigitalOutput(stDigitalOutput := stDigitalOutputData[7])
    Frame (768,164 660x110), invisible if: stDigitalOutputEmpty[8]
        shows SingleDigitalOutput(stDigitalOutput := stDigitalOutputData[8])
    Frame (768,274 660x110), invisible if: stDigitalOutputEmpty[9]
        shows SingleDigitalOutput(stDigitalOutput := stDigitalOutputData[9])
    Frame (768,384 660x110), invisible if: stDigitalOutputEmpty[10]
        shows SingleDigitalOutput(stDigitalOutput := stDigitalOutputData[10])
    Frame (768,494 660x110), invisible if: stDigitalOutputEmpty[11]
        shows SingleDigitalOutput(stDigitalOutput := stDigitalOutputData[11])
    Frame (768,604 660x110), invisible if: stDigitalOutputEmpty[12]
        shows SingleDigitalOutput(stDigitalOutput := stDigitalOutputData[12])
END_VISUALIZATION

// ---- VISUs/Pages/PageManualSafety.TcVIS
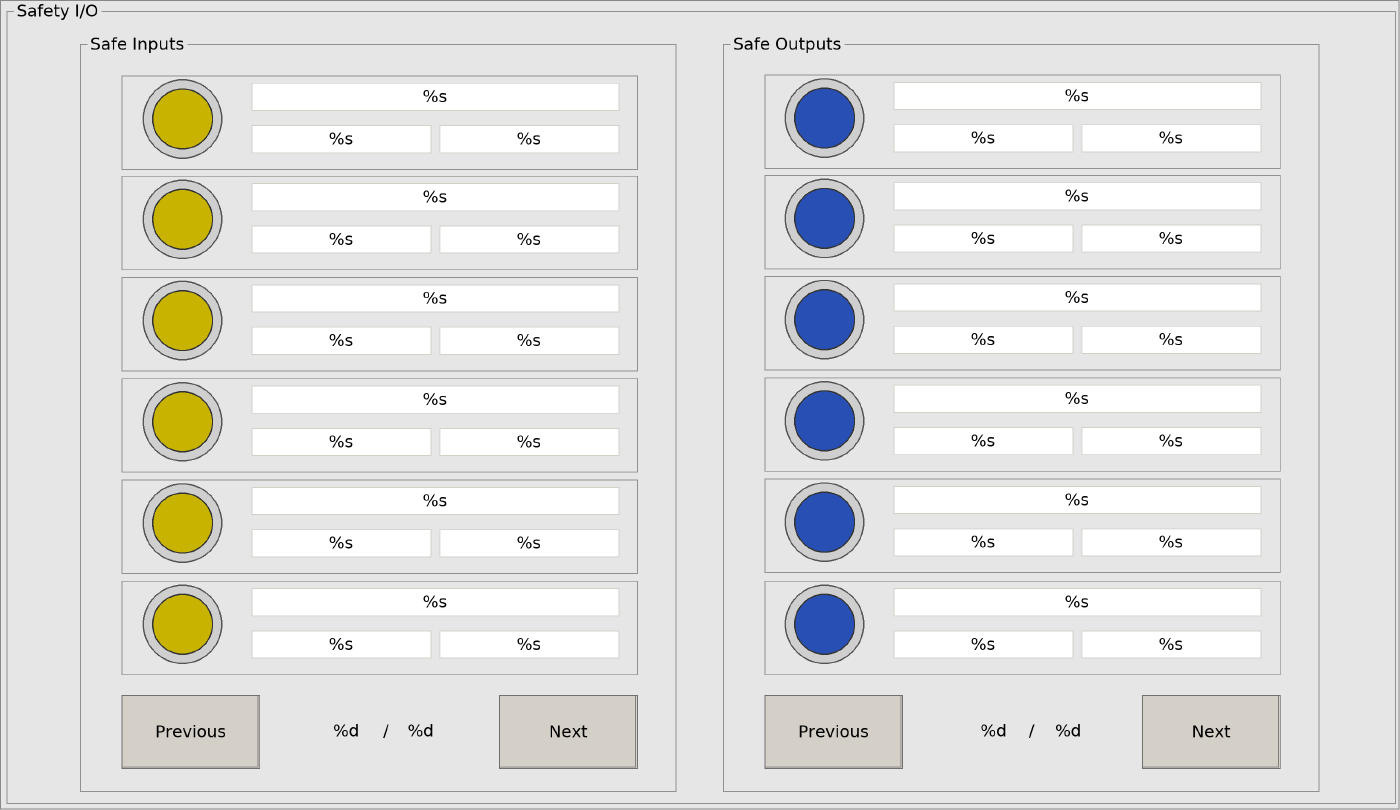
VISUALIZATION PageManualSafety  // 1520x880
VAR_IN_OUT
	btnNextInput			: BOOL;				(*  *)
	btnPreviousInput		: BOOL;				(*  *)
	btnNextOutput			: BOOL;				(*  *)
	btnPreviousOutput		: BOOL;				(*  *)
	
	bNextInvisibleInput		: BOOL;				(*  *)
	bPreviousInvisibleInput	: BOOL;				(*  *)
	bNextInvisibleOutput	: BOOL;				(*  *)
	bPreviousInvisibleOutput: BOOL;				(*  *)	
	
	iSafeInputSelectedPageIndex		: USINT;
	iSafeInputTotalPageIndex 		: USINT;
	iSafeOutputSelectedPageIndex	: USINT;
	iSafeOutputTotalPageIndex 		: USINT;
	
	stSafeOutputEmpty		: ARRAY[1..6] OF BOOL;
	stSafeOutputData		: ARRAY[1..6] OF ST_VisuCtrlOutputFrame;
	stSafeInputEmpty		: ARRAY[1..6] OF BOOL;
	stSafeInputData			: ARRAY[1..6] OF ST_VisuCtrlInputFrame;
END_VAR
    GroupBox (7,4 1508x869), "Safety I/O"
        GroupBox (80,36 647x820), "Safe Inputs"
            Frame (45,583 560x110), invisible if: stSafeInputEmpty[6]
                shows SingleSafeInput(stDigitalInput := stSafeInputData[6])
            Rectangle (345,729 50x50), "%d", text variable: iSafeInputTotalPageIndex+1
            Rectangle (264,729 50x50), "%d", text variable: iSafeInputSelectedPageIndex+1
            Rectangle (1461,1588 130x50), "/"
            Button (45,715 150x80), "Previous", pressed state: btnPreviousInput, invisible if: bPreviousInvisibleInput
                tap btnPreviousInput
            Button (455,715 150x80), "Next", pressed state: btnNextInput, invisible if: bNextInvisibleInput
                tap btnNextInput
            Frame (45,473 560x110), invisible if: stSafeInputEmpty[5]
                shows SingleSafeInput(stDigitalInput := stSafeInputData[5])
            Frame (45,363 560x110), invisible if: stSafeInputEmpty[4]
                shows SingleSafeInput(stDigitalInput := stSafeInputData[4])
            Frame (45,253 560x110), invisible if: stSafeInputEmpty[3]
                shows SingleSafeInput(stDigitalInput := stSafeInputData[3])
            Frame (45,143 560x110), invisible if: stSafeInputEmpty[2]
                shows SingleSafeInput(stDigitalInput := stSafeInputData[2])
            Frame (45,34 560x110), invisible if: stSafeInputEmpty[1]
                shows SingleSafeInput(stDigitalInput := stSafeInputData[1])
            Rectangle (267,729 130x50), "/"
        GroupBox (778,36 647x820), "Safe Outputs"
            Frame (45,583 560x110), invisible if: stSafeOutputEmpty[6]
                shows SingleSafeOutput(stDigitalOutput := stSafeOutputData[6])
            Rectangle (350,729 50x50), "%d", text variable: iSafeOutputTotalPageIndex+1
            Rectangle (269,729 50x50), "%d", text variable: iSafeOutputSelectedPageIndex+1
            Button (45,715 150x80), "Previous", pressed state: btnPreviousOutput, invisible if: bPreviousInvisibleOutput
                tap btnPreviousOutput
            Button (455,715 150x80), "Next", pressed state: btnNextOutput, invisible if: bNextInvisibleOutput
                tap btnNextOutput
            Frame (45,472 560x110), invisible if: stSafeOutputEmpty[5]
                shows SingleSafeOutput(stDigitalOutput := stSafeOutputData[5])
            Frame (45,362 560x110), invisible if: stSafeOutputEmpty[4]
                shows SingleSafeOutput(stDigitalOutput := stSafeOutputData[4])
            Frame (45,252 560x110), invisible if: stSafeOutputEmpty[3]
                shows SingleSafeOutput(stDigitalOutput := stSafeOutputData[3])
            Frame (45,142 560x110), invisible if: stSafeOutputEmpty[2]
                shows SingleSafeOutput(stDigitalOutput := stSafeOutputData[2])
            Frame (45,33 560x110), invisible if: stSafeOutputEmpty[1]
                shows SingleSafeOutput(stDigitalOutput := stSafeOutputData[1])
            Rectangle (270,729 130x50), "/"
END_VISUALIZATION

// ---- VISUs/Single/SingleCylinder.TcVIS
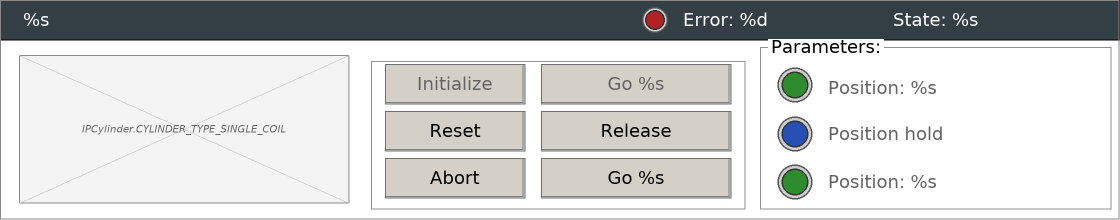
VISUALIZATION SingleCylinder  // 1120x220
VAR_IN_OUT
	stCylinder : ST_VisuCtrlCylinderFrame;
END_VAR
    Rectangle (0,0 1120x40)
    Textfield (20,5 524x30), "%s", text variable: stCylinder.sName
    Textfield (890,5 225x30), "State: %s", text list: 'TL_SingleCylinderState', text index: stCylinder.eCylinderState
    Lamp1 (640,5 30x30), variable: stCylinder.bError, style: Lamp-Lamp1-Red
    Textfield (680,5 200x30), "Error: %d", text variable: stCylinder.iErrorID
    GroupBox (760,39 351x170), "Parameters:"
        Rectangle (65,85 270x20), "Position hold", text variable: stCylinder.sHomeDescription
        Lamp1 (15,75 40x40), variable: stCylinder.bPositionHold, style: Lamp-Lamp1-Blue
        Rectangle (65,133 270x20), "Position: %s", text variable: stCylinder.sHomeDescription
        Rectangle (65,39 270x20), "Position: %s", text variable: stCylinder.sActiveDescription
        Lamp1 (15,26 40x40), variable: stCylinder.bSensorActive, style: Lamp-Lamp1-Green
        Lamp1 (15,123 40x40), variable: stCylinder.bSensorHome, style: Lamp-Lamp1-Green
    GroupBox (371,53 374x156)
        Button (170,105 190x40), "Go %s", text variable: stCylinder.sHomeDescription
            tap stCylinder.btnGoHome
        Button (170,58 190x40), "Release"
            tap stCylinder.btnRealase
        Button (170,11 190x40), "Go %s", text variable: stCylinder.sActiveDescription
            tap stCylinder.btnGoActive
        Button (14,105 140x40), "Abort", text variable: stCylinder.sHomeDescription
            tap stCylinder.btnAbort
        Button (14,58 140x40), "Reset"
            tap stCylinder.btnReset
        Button (14,11 140x40), "Initialize", text variable: stCylinder.sActiveDescription
            tap stCylinder.btnInit
    Image (19,55 330x148), image: IPCylinder.CYLINDER_TYPE_SINGLE_COIL
        p84334746: stCylinder.sCylinderImage
END_VISUALIZATION

// ---- VISUs/Single/SingleDigitalInput.TcVIS
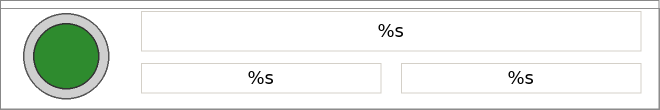
VISUALIZATION SingleDigitalInput  // 660x110
VAR_IN_OUT
	stDigitalInput : ST_VisuCtrlInputFrame;
END_VAR
    GroupBox (0,0 660x110)
        Lamp1 (16,6 100x100), variable: stDigitalInput.bIn, style: Lamp-Lamp1-Green
        Textfield (141,11 500x40), "%s", text variable: stDigitalInput.sName
        Textfield (141,63 240x30), "%s", text variable: stDigitalInput.sModuleType
        Textfield (401,63 240x30), "%s", text variable: stDigitalInput.sPortID
END_VISUALIZATION

// ---- VISUs/Single/SingleDigitalOutput.TcVIS
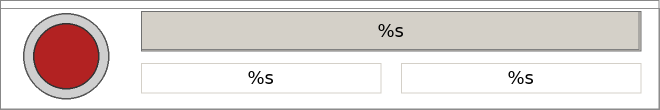
VISUALIZATION SingleDigitalOutput  // 660x110
VAR_IN_OUT
	stDigitalOutput : ST_VisuCtrlOutputFrame;
END_VAR
    GroupBox (0,0 660x110)
        Lamp1 (16,6 100x100), variable: stDigitalOutput.bOut, style: Lamp-Lamp1-Red
        Button (141,11 500x40), "%s", text variable: stDigitalOutput.sName, input disabled if: stDigitalOutput.bControlable, text list: ''
            toggle stDigitalOutput.btnOut
        Textfield (141,63 240x30), "%s", text variable: stDigitalOutput.sModuleType
        Textfield (401,63 240x30), "%s", text variable: stDigitalOutput.sPortID
END_VISUALIZATION

// ---- VISUs/Single/SingleSafeInput.TcVIS
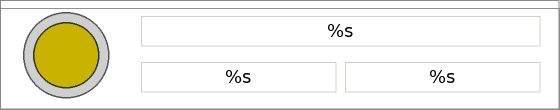
VISUALIZATION SingleSafeInput  // 560x110
VAR_IN_OUT
	stDigitalInput : ST_VisuCtrlInputFrame;
END_VAR
    GroupBox (0,0 560x110)
        Lamp1 (16,5 100x100), variable: stDigitalInput.bIn, style: Lamp-Lamp1-Yellow
        Textfield (141,16 399x30), "%s", text variable: stDigitalInput.sName
        Textfield (345,62 195x30), "%s", text variable: stDigitalInput.sPortID
        Textfield (141,62 195x30), "%s", text variable: stDigitalInput.sModuleType
END_VISUALIZATION

// ---- VISUs/Single/SingleSafeOutput.TcVIS
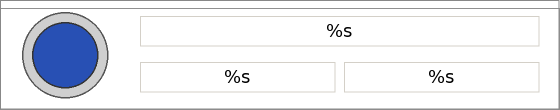
VISUALIZATION SingleSafeOutput  // 560x110
VAR_IN_OUT
	stDigitalOutput : ST_VisuCtrlOutputFrame;
END_VAR
    GroupBox (0,0 560x110)
        Lamp1 (15,5 100x100), variable: stDigitalOutput.bOut, style: Lamp-Lamp1-Blue
        Textfield (344,62 195x30), "%s", text variable: stDigitalOutput.sPortID
        Textfield (140,62 195x30), "%s", text variable: stDigitalOutput.sModuleType
        Textfield (140,16 399x30), "%s", text variable: stDigitalOutput.sName
END_VISUALIZATION

// ---- VISUs/Text Lists/TL_SingleCylinderState.TcTLO
TEXTLIST TL_SingleCylinderState
  0 = 'Uninitialized'
  10 = 'Initializing'
  20 = 'Ready initialized'
  30 = 'Idle'
  40 = 'Go active'
  50 = 'Go active done'
  60 = 'Go home'
  70 = 'Go home done'
  80 = 'Release'
  90 = 'Release done'
  100 = 'Reset'
  110 = 'Reset done'
  -10 = 'Aborting'
   = ''
END_TEXTLIST
